LIN {X 0,Y 395.166,Z 181.617,A -85,B 0,C 180,E1 13885.717,E2 13885.717} C_VEL
LIN {X 0,Y 390.867,Z 176.537,A -85,B 0,C 180,E1 13884.321,E2 13884.321} C_VEL
LIN {X 0,Y 388.966,Z 174.114,A -85,B 0,C 180,E1 13883.48,E2 13883.48} C_VEL
LIN {X 0,Y 387.756,Z 171.488,A -85,B 0,C 180,E1 13882.594,E2 13882.594} C_VEL
LIN {X 0,Y 385.429,Z 168.178,A -85,B 0,C 180,E1 13881.136,E2 13881.136} C_VEL
LIN {X 0,Y 384.536,Z 166.163,A -85,B 0,C 180,E1 13880.391,E2 13880.391} C_VEL
LIN {X 0,Y 381.955,Z 162.76,A -85,B 0,C 180,E1 13878.624,E2 13878.624} C_VEL
LIN {X 0,Y 381.043,Z 160.578,A -85,B 0,C 180,E1 13877.721,E2 13877.721} C_VEL
LIN {X 0,Y 378.363,Z 157.325,A -85,B 0,C 180,E1 13875.637,E2 13875.637} C_VEL
LIN {X 0,Y 377.709,Z 155.286,A -85,B 0,C 180,E1 13874.565,E2 13874.565} C_VEL
LIN {X 0,Y 377.671,Z 154.998,A -85,B 0,C 180,E1 13871.762,E2 13871.762} C_VEL
LIN {X 0,Y 377.67,Z 154.99,A -85,B 0,C 180,E1 13867.759,E2 13867.759} C_VEL
LIN {X 0,Y 377.664,Z 154.988,A -85,B 0,C 180,E1 13863.795,E2 13863.795} C_VEL
LIN {X 0,Y 377.658,Z 154.987,A -85,B 0,C 180,E1 13859.848,E2 13859.848} C_VEL
LIN {X 0,Y 377.652,Z 154.988,A -85,B 0,C 180,E1 13855.901,E2 13855.901} C_VEL
LIN {X 0,Y 377.647,Z 154.992,A -85,B 0,C 180,E1 13851.933,E2 13851.933} C_VEL
LIN {X 0,Y 377.647,Z 154.999,A -85,B 0,C 180,E1 13847.927,E2 13847.927} C_VEL
LIN {X 0,Y 377.644,Z 155.008,A -85,B 0,C 180,E1 13843.958,E2 13843.958} C_VEL
LIN {X 0,Y 377.723,Z 155.416,A -85,B 0,C 180,E1 13842.855,E2 13842.855} C_VEL
LIN {X 0,Y 379.411,Z 159.029,A -85,B 0,C 180,E1 13840.927,E2 13840.927} C_VEL
LIN {X 0,Y 381.432,Z 161.353,A -85,B 0,C 180,E1 13839.435,E2 13839.435} C_VEL
LIN {X 0,Y 383.122,Z 164.838,A -85,B 0,C 180,E1 13837.926,E2 13837.926} C_VEL
LIN {X 0,Y 384.74,Z 166.714,A -85,B 0,C 180,E1 13836.895,E2 13836.895} C_VEL
LIN {X 0,Y 386.737,Z 170.482,A -85,B 0,C 180,E1 13835.402,E2 13835.402} C_VEL
LIN {X 0,Y 387.954,Z 172.11,A -85,B 0,C 180,E1 13834.67,E2 13834.67} C_VEL
LIN {X 0,Y 390.476,Z 176.478,A -85,B 0,C 180,E1 13833.049,E2 13833.049} C_VEL
LIN {X 0,Y 394.111,Z 183.067,A -85,B 0,C 180,E1 13830.849,E2 13830.849} C_VEL
LIN {X 0,Y 396.955,Z 188.298,A -85,B 0,C 180,E1 13829.248,E2 13829.248} C_VEL
LIN {X 0,Y 401.414,Z 196.48,A -85,B 0,C 180,E1 13826.941,E2 13826.941} C_VEL
LIN {X 0,Y 408.691,Z 206.89,A -85,B 0,C 180,E1 13824.863,E2 13824.863} C_VEL
LIN {X 0,Y 417.567,Z 219.734,A -85,B 0,C 180,E1 13822.627,E2 13822.627} C_VEL
LIN {X 0,Y 427.427,Z 235.069,A -85,B 0,C 180,E1 13820.355,E2 13820.355} C_VEL
LIN {X 0,Y 431.676,Z 242.453,A -85,B 0,C 180,E1 13819.423,E2 13819.423} C_VEL
LIN {X 0,Y 432.974,Z 254.438,A -85,B 0,C 180,E1 13818.9,E2 13818.9} C_VEL
LIN {X 0,Y 424.415,Z 482.924,A -85,B 0,C 180,E1 13814.793,E2 13814.793} C_VEL
LIN {X 0,Y 422.877,Z 518.615,A -85,B 0,C 180,E1 13814.119,E2 13814.119} C_VEL
LIN {X 0,Y 420.953,Z 540.04,A -85,B 0,C 180,E1 13813.517,E2 13813.517} C_VEL
LIN {X 0,Y 418.413,Z 561.095,A -85,B 0,C 180,E1 13812.691,E2 13812.691} C_VEL
LIN {X 0,Y 415.519,Z 580.617,A -85,B 0,C 180,E1 13811.707,E2 13811.707} C_VEL
LIN {X 0,Y 412.005,Z 600.005,A -85,B 0,C 180,E1 13810.478,E2 13810.478} C_VEL
LIN {X 0,Y 408.151,Z 618.986,A -85,B 0,C 180,E1 13809.018,E2 13809.018} C_VEL
LIN {X 0,Y 404.015,Z 637.17,A -85,B 0,C 180,E1 13807.323,E2 13807.323} C_VEL
LIN {X 0,Y 399.701,Z 654.729,A -85,B 0,C 180,E1 13805.363,E2 13805.363} C_VEL
LIN {X 0,Y 395.442,Z 671.248,A -85,B 0,C 180,E1 13803.183,E2 13803.183} C_VEL
LIN {X 0,Y 392.212,Z 683.238,A -85,B 0,C 180,E1 13801.325,E2 13801.325} C_VEL
LIN {X 0,Y 389.972,Z 688.467,A -85,B 0,C 180,E1 13800.537,E2 13800.537} C_VEL
LIN {X 0,Y 381.254,Z 701.209,A -85,B 0,C 180,E1 13798.63,E2 13798.63} C_VEL
LIN {X 0,Y 379.092,Z 705.741,A -85,B 0,C 180,E1 13797.739,E2 13797.739} C_VEL
LIN {X 0,Y 375.806,Z 717.722,A -85,B 0,C 180,E1 13794.857,E2 13794.857} C_VEL
LIN {X 0,Y 373.033,Z 728.698,A -85,B 0,C 180,E1 13791.708,E2 13791.708} C_VEL
LIN {X 0,Y 370.991,Z 737.873,A -85,B 0,C 180,E1 13788.543,E2 13788.543} C_VEL
LIN {X 0,Y 369.523,Z 745.565,A -85,B 0,C 180,E1 13785.216,E2 13785.216} C_VEL
LIN {X 0,Y 368.595,Z 751.959,A -85,B 0,C 180,E1 13781.69,E2 13781.69} C_VEL
LIN {X 0,Y 368.168,Z 756.552,A -85,B 0,C 180,E1 13778.275,E2 13778.275} C_VEL
LIN {X 0,Y 367.989,Z 759.37,A -85,B 0,C 180,E1 13774.988,E2 13774.988} C_VEL
LIN {X 0,Y 367.942,Z 760.876,A -85,B 0,C 180,E1 13771.557,E2 13771.557} C_VEL
LIN {X 0,Y 367.948,Z 760.909,A -85,B 0,C 180,E1 13768.599,E2 13768.599} C_VEL
LIN {X 0,Y 367.986,Z 759.541,A -85,B 0,C 180,E1 13765.168,E2 13765.168} C_VEL
LIN {X 0,Y 368.12,Z 756.942,A -85,B 0,C 180,E1 13762.038,E2 13762.038} C_VEL
LIN {X 0,Y 368.533,Z 752.507,A -85,B 0,C 180,E1 13758.577,E2 13758.577} C_VEL
LIN {X 0,Y 369.344,Z 746.768,A -85,B 0,C 180,E1 13755.258,E2 13755.258} C_VEL
LIN {X 0,Y 370.692,Z 739.255,A -85,B 0,C 180,E1 13751.93,E2 13751.93} C_VEL
LIN {X 0,Y 372.772,Z 729.787,A -85,B 0,C 180,E1 13748.55,E2 13748.55} C_VEL
LIN {X 0,Y 375.424,Z 719.28,A -85,B 0,C 180,E1 13745.452,E2 13745.452} C_VEL
LIN {X 0,Y 378.7,Z 707.114,A -85,B 0,C 180,E1 13742.482,E2 13742.482} C_VEL
LIN {X 0,Y 382.493,Z 693.534,A -85,B 0,C 180,E1 13739.702,E2 13739.702} C_VEL
LIN {X 0,Y 386.623,Z 679.075,A -85,B 0,C 180,E1 13737.193,E2 13737.193} C_VEL
LIN {X 0,Y 390.999,Z 663.173,A -85,B 0,C 180,E1 13734.876,E2 13734.876} C_VEL
LIN {X 0,Y 395.564,Z 645.973,A -85,B 0,C 180,E1 13732.771,E2 13732.771} C_VEL
LIN {X 0,Y 399.96,Z 628.38,A -85,B 0,C 180,E1 13730.953,E2 13730.953} C_VEL
LIN {X 0,Y 404.219,Z 609.241,A -85,B 0,C 180,E1 13729.325,E2 13729.325} C_VEL
LIN {X 0,Y 408.257,Z 588.889,A -85,B 0,C 180,E1 13727.909,E2 13727.909} C_VEL
LIN {X 0,Y 411.78,Z 568.3,A -85,B 0,C 180,E1 13726.756,E2 13726.756} C_VEL
LIN {X 0,Y 414.498,Z 548.215,A -85,B 0,C 180,E1 13725.889,E2 13725.889} C_VEL
LIN {X 0,Y 416.821,Z 526.068,A -85,B 0,C 180,E1 13725.177,E2 13725.177} C_VEL
LIN {X 0,Y 418.288,Z 503.726,A -85,B 0,C 180,E1 13724.681,E2 13724.681} C_VEL
LIN {X 0,Y 426.979,Z 279.836,A -85,B 0,C 180,E1 13720.629,E2 13720.629} C_VEL
LIN {X 0,Y 427.951,Z 254.162,A -85,B 0,C 180,E1 13720.132,E2 13720.132} C_VEL
LIN {X 0,Y 426.916,Z 246.348,A -85,B 0,C 180,E1 13719.746,E2 13719.746} C_VEL
LIN {X 0,Y 417.063,Z 230.424,A -85,B 0,C 180,E1 13717.469,E2 13717.469} C_VEL
LIN {X 0,Y 407.725,Z 216.316,A -85,B 0,C 180,E1 13715.104,E2 13715.104} C_VEL
LIN {X 0,Y 397.968,Z 202.523,A -85,B 0,C 180,E1 13712.354,E2 13712.354} C_VEL
LIN {X 0,Y 392.606,Z 195.303,A -85,B 0,C 180,E1 13710.62,E2 13710.62} C_VEL
LIN {X 0,Y 390.03,Z 190.525,A -85,B 0,C 180,E1 13709.149,E2 13709.149} C_VEL
LIN {X 0,Y 387.794,Z 186.527,A -85,B 0,C 180,E1 13707.819,E2 13707.819} C_VEL
LIN {X 0,Y 385.711,Z 182.654,A -85,B 0,C 180,E1 13706.479,E2 13706.479} C_VEL
LIN {X 0,Y 382.811,Z 177.599,A -85,B 0,C 180,E1 13704.538,E2 13704.538} C_VEL
LIN {X 0,Y 380.501,Z 173.731,A -85,B 0,C 180,E1 13702.887,E2 13702.887} C_VEL
LIN {X 0,Y 379.69,Z 172.421,A -85,B 0,C 180,E1 13702.285,E2 13702.285} C_VEL
LIN {X 0,Y 377.515,Z 169.146,A -85,B 0,C 180,E1 13700.625,E2 13700.625} C_VEL
LIN {X 0,Y 376.786,Z 167.346,A -85,B 0,C 180,E1 13699.857,E2 13699.857} C_VEL
LIN {X 0,Y 373.937,Z 163.505,A -85,B 0,C 180,E1 13697.426,E2 13697.426} C_VEL
LIN {X 0,Y 373.044,Z 161.554,A -85,B 0,C 180,E1 13696.346,E2 13696.346} C_VEL
LIN {X 0,Y 370.204,Z 157.928,A -85,B 0,C 180,E1 13693.272,E2 13693.272} C_VEL
LIN {X 0,Y 369.725,Z 156.173,A -85,B 0,C 180,E1 13691.861,E2 13691.861} C_VEL
LIN {X 0,Y 369.703,Z 155.98,A -85,B 0,C 180,E1 13687.928,E2 13687.928} C_VEL
LIN {X 0,Y 369.705,Z 155.977,A -85,B 0,C 180,E1 13683.877,E2 13683.877} C_VEL
LIN {X 0,Y 369.708,Z 155.977,A -85,B 0,C 180,E1 13679.845,E2 13679.845} C_VEL
LIN {X 0,Y 369.712,Z 155.982,A -85,B 0,C 180,E1 13675.657,E2 13675.657} C_VEL
LIN {X 0,Y 369.717,Z 155.989,A -85,B 0,C 180,E1 13671.603,E2 13671.603} C_VEL
LIN {X 0,Y 369.788,Z 156.38,A -85,B 0,C 180,E1 13670.192,E2 13670.192} C_VEL
LIN {X 0,Y 371.857,Z 160.462,A -85,B 0,C 180,E1 13667.105,E2 13667.105} C_VEL
LIN {X 0,Y 373.69,Z 162.433,A -85,B 0,C 180,E1 13665.433,E2 13665.433} C_VEL
LIN {X 0,Y 375.581,Z 166.123,A -85,B 0,C 180,E1 13663.45,E2 13663.45} C_VEL
LIN {X 0,Y 377.214,Z 167.9,A -85,B 0,C 180,E1 13662.253,E2 13662.253} C_VEL
LIN {X 0,Y 379.311,Z 171.902,A -85,B 0,C 180,E1 13660.442,E2 13660.442} C_VEL
LIN {X 0,Y 380.668,Z 173.567,A -85,B 0,C 180,E1 13659.554,E2 13659.554} C_VEL
LIN {X 0,Y 382.518,Z 176.962,A -85,B 0,C 180,E1 13658.293,E2 13658.293} C_VEL
LIN {X 0,Y 385.014,Z 179.629,A -85,B 0,C 180,E1 13657.357,E2 13657.357} C_VEL
LIN {X 0,Y 390.258,Z 185.827,A -85,B 0,C 180,E1 13655.518,E2 13655.518} C_VEL
LIN {X 0,Y 394.878,Z 191.397,A -85,B 0,C 180,E1 13654.021,E2 13654.021} C_VEL
LIN {X 0,Y 399.491,Z 197.171,A -85,B 0,C 180,E1 13652.62,E2 13652.62} C_VEL
LIN {X 0,Y 406.598,Z 206.189,A -85,B 0,C 180,E1 13650.621,E2 13650.621} C_VEL
LIN {X 0,Y 417.605,Z 221.402,A -85,B 0,C 180,E1 13647.811,E2 13647.811} C_VEL
LIN {X 0,Y 428.267,Z 237.38,A -85,B 0,C 180,E1 13645.355,E2 13645.355} C_VEL
LIN {X 0,Y 431.593,Z 243.039,A -85,B 0,C 180,E1 13644.622,E2 13644.622} C_VEL
LIN {X 0,Y 421.696,Z 453.338,A -85,B 0,C 180,E1 13640.539,E2 13640.539} C_VEL
LIN {X 0,Y 418.781,Z 513.038,A -85,B 0,C 180,E1 13639.345,E2 13639.345} C_VEL
LIN {X 0,Y 416.496,Z 536.285,A -85,B 0,C 180,E1 13638.676,E2 13638.676} C_VEL
LIN {X 0,Y 413.464,Z 560.266,A -85,B 0,C 180,E1 13637.728,E2 13637.728} C_VEL
LIN {X 0,Y 410.168,Z 581.646,A -85,B 0,C 180,E1 13636.637,E2 13636.637} C_VEL
LIN {X 0,Y 406.403,Z 602.444,A -85,B 0,C 180,E1 13635.316,E2 13635.316} C_VEL
LIN {X 0,Y 402.384,Z 622.536,A -85,B 0,C 180,E1 13633.789,E2 13633.789} C_VEL
LIN {X 0,Y 398.064,Z 641.897,A -85,B 0,C 180,E1 13632.019,E2 13632.019} C_VEL
LIN {X 0,Y 393.619,Z 660.879,A -85,B 0,C 180,E1 13629.989,E2 13629.989} C_VEL
LIN {X 0,Y 389.314,Z 678.385,A -85,B 0,C 180,E1 13627.771,E2 13627.771} C_VEL
LIN {X 0,Y 384.71,Z 696.784,A -85,B 0,C 180,E1 13625.047,E2 13625.047} C_VEL
LIN {X 0,Y 380.795,Z 712.759,A -85,B 0,C 180,E1 13622.277,E2 13622.277} C_VEL
LIN {X 0,Y 377.294,Z 727.194,A -85,B 0,C 180,E1 13619.323,E2 13619.323} C_VEL
LIN {X 0,Y 374.329,Z 740.523,A -85,B 0,C 180,E1 13616.149,E2 13616.149} C_VEL
LIN {X 0,Y 372.125,Z 751.393,A -85,B 0,C 180,E1 13613.096,E2 13613.096} C_VEL
LIN {X 0,Y 370.27,Z 762.065,A -85,B 0,C 180,E1 13609.538,E2 13609.538} C_VEL
LIN {X 0,Y 369.201,Z 769.556,A -85,B 0,C 180,E1 13606.52,E2 13606.52} C_VEL
LIN {X 0,Y 368.446,Z 776.529,A -85,B 0,C 180,E1 13603.017,E2 13603.017} C_VEL
LIN {X 0,Y 368.102,Z 781.139,A -85,B 0,C 180,E1 13600.011,E2 13600.011} C_VEL
LIN {X 0,Y 367.961,Z 784.976,A -85,B 0,C 180,E1 13596.553,E2 13596.553} C_VEL
LIN {X 0,Y 367.926,Z 786.994,A -85,B 0,C 180,E1 13593.427,E2 13593.427} C_VEL
LIN {X 0,Y 367.923,Z 787.81,A -85,B 0,C 180,E1 13590.311,E2 13590.311} C_VEL
LIN {X 0,Y 367.929,Z 787.138,A -85,B 0,C 180,E1 13586.884,E2 13586.884} C_VEL
LIN {X 0,Y 367.952,Z 785.218,A -85,B 0,C 180,E1 13583.76,E2 13583.76} C_VEL
LIN {X 0,Y 368.083,Z 781.58,A -85,B 0,C 180,E1 13580.305,E2 13580.305} C_VEL
LIN {X 0,Y 368.403,Z 777.077,A -85,B 0,C 180,E1 13577.301,E2 13577.301} C_VEL
LIN {X 0,Y 369.11,Z 770.303,A -85,B 0,C 180,E1 13573.799,E2 13573.799} C_VEL
LIN {X 0,Y 370.21,Z 762.431,A -85,B 0,C 180,E1 13570.598,E2 13570.598} C_VEL
LIN {X 0,Y 372.028,Z 751.939,A -85,B 0,C 180,E1 13567.065,E2 13567.065} C_VEL
LIN {X 0,Y 374.196,Z 741.127,A -85,B 0,C 180,E1 13564.011,E2 13564.011} C_VEL
LIN {X 0,Y 377.16,Z 727.779,A -85,B 0,C 180,E1 13560.806,E2 13560.806} C_VEL
LIN {X 0,Y 380.715,Z 713.082,A -85,B 0,C 180,E1 13557.784,E2 13557.784} C_VEL
LIN {X 0,Y 384.475,Z 697.69,A -85,B 0,C 180,E1 13555.102,E2 13555.102} C_VEL
LIN {X 0,Y 388.899,Z 680.083,A -85,B 0,C 180,E1 13552.46,E2 13552.46} C_VEL
LIN {X 0,Y 393.143,Z 662.726,A -85,B 0,C 180,E1 13550.237,E2 13550.237} C_VEL
LIN {X 0,Y 397.724,Z 643.281,A -85,B 0,C 180,E1 13548.121,E2 13548.121} C_VEL
LIN {X 0,Y 402.194,Z 623.378,A -85,B 0,C 180,E1 13546.283,E2 13546.283} C_VEL
LIN {X 0,Y 406.231,Z 603.236,A -85,B 0,C 180,E1 13544.743,E2 13544.743} C_VEL
LIN {X 0,Y 410.06,Z 582.206,A -85,B 0,C 180,E1 13543.398,E2 13543.398} C_VEL
LIN {X 0,Y 413.347,Z 560.902,A -85,B 0,C 180,E1 13542.305,E2 13542.305} C_VEL
LIN {X 0,Y 416.458,Z 536.382,A -85,B 0,C 180,E1 13541.331,E2 13541.331} C_VEL
LIN {X 0,Y 418.745,Z 513.127,A -85,B 0,C 180,E1 13540.661,E2 13540.661} C_VEL
LIN {X 0,Y 421.719,Z 452.113,A -85,B 0,C 180,E1 13539.441,E2 13539.441} C_VEL
LIN {X 0,Y 431.558,Z 242.837,A -85,B 0,C 180,E1 13535.378,E2 13535.378} C_VEL
LIN {X 0,Y 423.08,Z 229.475,A -85,B 0,C 180,E1 13533.492,E2 13533.492} C_VEL
LIN {X 0,Y 413.033,Z 214.984,A -85,B 0,C 180,E1 13531.079,E2 13531.079} C_VEL
LIN {X 0,Y 404.563,Z 203.689,A -85,B 0,C 180,E1 13528.852,E2 13528.852} C_VEL
LIN {X 0,Y 397.353,Z 194.401,A -85,B 0,C 180,E1 13526.77,E2 13526.77} C_VEL
LIN {X 0,Y 392.396,Z 188.417,A -85,B 0,C 180,E1 13525.224,E2 13525.224} C_VEL
LIN {X 0,Y 388.174,Z 183.385,A -85,B 0,C 180,E1 13523.813,E2 13523.813} C_VEL
LIN {X 0,Y 383.503,Z 177.934,A -85,B 0,C 180,E1 13522.131,E2 13522.131} C_VEL
LIN {X 0,Y 381.462,Z 175.518,A -85,B 0,C 180,E1 13521.205,E2 13521.205} C_VEL
LIN {X 0,Y 380.181,Z 172.78,A -85,B 0,C 180,E1 13520.152,E2 13520.152} C_VEL
LIN {X 0,Y 377.689,Z 169.301,A -85,B 0,C 180,E1 13518.362,E2 13518.362} C_VEL
LIN {X 0,Y 376.74,Z 167.247,A -85,B 0,C 180,E1 13517.451,E2 13517.451} C_VEL
LIN {X 0,Y 374.184,Z 163.875,A -85,B 0,C 180,E1 13515.339,E2 13515.339} C_VEL
LIN {X 0,Y 373.131,Z 161.609,A -85,B 0,C 180,E1 13514.113,E2 13514.113} C_VEL
LIN {X 0,Y 370.333,Z 158.146,A -85,B 0,C 180,E1 13511.209,E2 13511.209} C_VEL
LIN {X 0,Y 369.759,Z 156.148,A -85,B 0,C 180,E1 13509.651,E2 13509.651} C_VEL
LIN {X 0,Y 369.738,Z 155.984,A -85,B 0,C 180,E1 13505.586,E2 13505.586} C_VEL
LIN {X 0,Y 369.746,Z 155.991,A -85,B 0,C 180,E1 13501.394,E2 13501.394} C_VEL
LIN {X 0,Y 369.74,Z 155.982,A -85,B 0,C 180,E1 13497.365,E2 13497.365} C_VEL
LIN {X 0,Y 369.751,Z 155.974,A -85,B 0,C 180,E1 13493.166,E2 13493.166} C_VEL
LIN {X 0,Y 369.729,Z 155.975,A -85,B 0,C 180,E1 13489.002,E2 13489.002} C_VEL
LIN {X 0,Y 369.796,Z 156.421,A -85,B 0,C 180,E1 13487.508,E2 13487.508} C_VEL
LIN {X 0,Y 371.777,Z 160.439,A -85,B 0,C 180,E1 13484.558,E2 13484.558} C_VEL
LIN {X 0,Y 373.498,Z 162.115,A -85,B 0,C 180,E1 13483.034,E2 13483.034} C_VEL
LIN {X 0,Y 375.351,Z 165.9,A -85,B 0,C 180,E1 13481.018,E2 13481.018} C_VEL
LIN {X 0,Y 377.132,Z 167.939,A -85,B 0,C 180,E1 13479.677,E2 13479.677} C_VEL
LIN {X 0,Y 379.001,Z 171.688,A -85,B 0,C 180,E1 13477.999,E2 13477.999} C_VEL
LIN {X 0,Y 380.362,Z 173.32,A -85,B 0,C 180,E1 13477.104,E2 13477.104} C_VEL
LIN {X 0,Y 382.66,Z 177.433,A -85,B 0,C 180,E1 13475.405,E2 13475.405} C_VEL
LIN {X 0,Y 383.696,Z 179.193,A -85,B 0,C 180,E1 13474.7,E2 13474.7} C_VEL
LIN {X 0,Y 386.674,Z 184.421,A -85,B 0,C 180,E1 13472.762,E2 13472.762} C_VEL
LIN {X 0,Y 389.597,Z 189.698,A -85,B 0,C 180,E1 13470.984,E2 13470.984} C_VEL
LIN {X 0,Y 392.155,Z 194.438,A -85,B 0,C 180,E1 13469.51,E2 13469.51} C_VEL
LIN {X 0,Y 394.527,Z 198.004,A -85,B 0,C 180,E1 13468.571,E2 13468.571} C_VEL
LIN {X 0,Y 404.508,Z 211.689,A -85,B 0,C 180,E1 13465.65,E2 13465.65} C_VEL
LIN {X 0,Y 414.629,Z 226.73,A -85,B 0,C 180,E1 13463.011,E2 13463.011} C_VEL
LIN {X 0,Y 424.96,Z 243.09,A -85,B 0,C 180,E1 13460.582,E2 13460.582} C_VEL
LIN {X 0,Y 427.049,Z 247.02,A -85,B 0,C 180,E1 13460.105,E2 13460.105} C_VEL
LIN {X 0,Y 427.957,Z 256.049,A -85,B 0,C 180,E1 13459.711,E2 13459.711} C_VEL
LIN {X 0,Y 418.94,Z 484.862,A -85,B 0,C 180,E1 13455.564,E2 13455.564} C_VEL
LIN {X 0,Y 417.374,Z 518.914,A -85,B 0,C 180,E1 13454.911,E2 13454.911} C_VEL
LIN {X 0,Y 415.369,Z 540.34,A -85,B 0,C 180,E1 13454.304,E2 13454.304} C_VEL
LIN {X 0,Y 412.717,Z 561.358,A -85,B 0,C 180,E1 13453.472,E2 13453.472} C_VEL
LIN {X 0,Y 409.609,Z 581.469,A -85,B 0,C 180,E1 13452.448,E2 13452.448} C_VEL
LIN {X 0,Y 405.956,Z 600.706,A -85,B 0,C 180,E1 13451.21,E2 13451.21} C_VEL
LIN {X 0,Y 401.753,Z 620.373,A -85,B 0,C 180,E1 13449.668,E2 13449.668} C_VEL
LIN {X 0,Y 397.464,Z 638.443,A -85,B 0,C 180,E1 13447.955,E2 13447.955} C_VEL
LIN {X 0,Y 393.006,Z 655.66,A -85,B 0,C 180,E1 13445.992,E2 13445.992} C_VEL
LIN {X 0,Y 388.529,Z 672.159,A -85,B 0,C 180,E1 13443.769,E2 13443.769} C_VEL
LIN {X 0,Y 384.293,Z 687.21,A -85,B 0,C 180,E1 13441.356,E2 13441.356} C_VEL
LIN {X 0,Y 380.408,Z 700.921,A -85,B 0,C 180,E1 13438.749,E2 13438.749} C_VEL
LIN {X 0,Y 379.092,Z 705.741,A -85,B 0,C 180,E1 13437.739,E2 13437.739} C_VEL
LIN {X 0,Y 376.959,Z 710.119,A -85,B 0,C 180,E1 13436.816,E2 13436.816} C_VEL
LIN {X 0,Y 368.516,Z 720.971,A -85,B 0,C 180,E1 13434.547,E2 13434.547} C_VEL
LIN {X 0,Y 366.59,Z 724.682,A -85,B 0,C 180,E1 13433.538,E2 13433.538} C_VEL
LIN {X 0,Y 364.042,Z 734.721,A -85,B 0,C 180,E1 13430.246,E2 13430.246} C_VEL
LIN {X 0,Y 362.2,Z 743.207,A -85,B 0,C 180,E1 13426.849,E2 13426.849} C_VEL
LIN {X 0,Y 361.017,Z 749.841,A -85,B 0,C 180,E1 13423.452,E2 13423.452} C_VEL
LIN {X 0,Y 360.343,Z 755.12,A -85,B 0,C 180,E1 13419.906,E2 13419.906} C_VEL
LIN {X 0,Y 360.064,Z 758.667,A -85,B 0,C 180,E1 13416.537,E2 13416.537} C_VEL
LIN {X 0,Y 359.964,Z 760.664,A -85,B 0,C 180,E1 13413.185,E2 13413.185} C_VEL
LIN {X 0,Y 359.952,Z 761.37,A -85,B 0,C 180,E1 13409.823,E2 13409.823} C_VEL
LIN {X 0,Y 359.968,Z 760.573,A -85,B 0,C 180,E1 13406.497,E2 13406.497} C_VEL
LIN {X 0,Y 360.081,Z 758.301,A -85,B 0,C 180,E1 13402.982,E2 13402.982} C_VEL
LIN {X 0,Y 360.367,Z 754.841,A -85,B 0,C 180,E1 13399.772,E2 13399.772} C_VEL
LIN {X 0,Y 361.082,Z 749.428,A -85,B 0,C 180,E1 13396.224,E2 13396.224} C_VEL
LIN {X 0,Y 362.308,Z 742.685,A -85,B 0,C 180,E1 13392.826,E2 13392.826} C_VEL
LIN {X 0,Y 364.212,Z 734.045,A -85,B 0,C 180,E1 13389.413,E2 13389.413} C_VEL
LIN {X 0,Y 366.741,Z 724.114,A -85,B 0,C 180,E1 13386.204,E2 13386.204} C_VEL
LIN {X 0,Y 369.976,Z 712.627,A -85,B 0,C 180,E1 13383.104,E2 13383.104} C_VEL
LIN {X 0,Y 373.6,Z 700.227,A -85,B 0,C 180,E1 13380.324,E2 13380.324} C_VEL
LIN {X 0,Y 378.004,Z 685.418,A -85,B 0,C 180,E1 13377.524,E2 13377.524} C_VEL
LIN {X 0,Y 382.562,Z 670.106,A -85,B 0,C 180,E1 13375.085,E2 13375.085} C_VEL
LIN {X 0,Y 387.044,Z 654.195,A -85,B 0,C 180,E1 13372.963,E2 13372.963} C_VEL
LIN {X 0,Y 392.055,Z 635.422,A -85,B 0,C 180,E1 13370.863,E2 13370.863} C_VEL
LIN {X 0,Y 396.646,Z 616.823,A -85,B 0,C 180,E1 13369.134,E2 13369.134} C_VEL
LIN {X 0,Y 400.827,Z 597.451,A -85,B 0,C 180,E1 13367.663,E2 13367.663} C_VEL
LIN {X 0,Y 404.786,Z 576.315,A -85,B 0,C 180,E1 13366.364,E2 13366.364} C_VEL
LIN {X 0,Y 408.071,Z 555.322,A -85,B 0,C 180,E1 13365.347,E2 13365.347} C_VEL
LIN {X 0,Y 410.579,Z 534.464,A -85,B 0,C 180,E1 13364.597,E2 13364.597} C_VEL
LIN {X 0,Y 412.508,Z 511.375,A -85,B 0,C 180,E1 13364.013,E2 13364.013} C_VEL
LIN {X 0,Y 421.76,Z 287.062,A -85,B 0,C 180,E1 13359.904,E2 13359.904} C_VEL
LIN {X 0,Y 423.033,Z 255.87,A -85,B 0,C 180,E1 13359.304,E2 13359.304} C_VEL
LIN {X 0,Y 422.307,Z 250.816,A -85,B 0,C 180,E1 13359.034,E2 13359.034} C_VEL
LIN {X 0,Y 412.164,Z 234.313,A -85,B 0,C 180,E1 13356.596,E2 13356.596} C_VEL
LIN {X 0,Y 403.507,Z 221.329,A -85,B 0,C 180,E1 13354.314,E2 13354.314} C_VEL
LIN {X 0,Y 395.293,Z 209.44,A -85,B 0,C 180,E1 13351.914,E2 13351.914} C_VEL
LIN {X 0,Y 386.834,Z 198.228,A -85,B 0,C 180,E1 13349.158,E2 13349.158} C_VEL
LIN {X 0,Y 383.857,Z 193.883,A -85,B 0,C 180,E1 13347.96,E2 13347.96} C_VEL
LIN {X 0,Y 380.77,Z 188.523,A -85,B 0,C 180,E1 13346.01,E2 13346.01} C_VEL
LIN {X 0,Y 378.416,Z 184.172,A -85,B 0,C 180,E1 13344.343,E2 13344.343} C_VEL
LIN {X 0,Y 376.141,Z 180.315,A -85,B 0,C 180,E1 13342.671,E2 13342.671} C_VEL
LIN {X 0,Y 375.196,Z 178.887,A -85,B 0,C 180,E1 13341.973,E2 13341.973} C_VEL
LIN {X 0,Y 373.095,Z 175.329,A -85,B 0,C 180,E1 13340.225,E2 13340.225} C_VEL
LIN {X 0,Y 372.382,Z 173.915,A -85,B 0,C 180,E1 13339.538,E2 13339.538} C_VEL
LIN {X 0,Y 369.75,Z 170.073,A -85,B 0,C 180,E1 13337.143,E2 13337.143} C_VEL
LIN {X 0,Y 368.992,Z 168.429,A -85,B 0,C 180,E1 13336.207,E2 13336.207} C_VEL
LIN {X 0,Y 366.145,Z 164.537,A -85,B 0,C 180,E1 13332.94,E2 13332.94} C_VEL
LIN {X 0,Y 365.359,Z 162.745,A -85,B 0,C 180,E1 13331.524,E2 13331.524} C_VEL
LIN {X 0,Y 362.162,Z 158.598,A -85,B 0,C 180,E1 13324.275,E2 13324.275} C_VEL
LIN {X 0,Y 362.001,Z 157.968,A -85,B 0,C 180,E1 13320.633,E2 13320.633} C_VEL
LIN {X 0,Y 362.394,Z 159.146,A -85,B 0,C 180,E1 13316.837,E2 13316.837} C_VEL
LIN {X 0,Y 365.714,Z 163.154,A -85,B 0,C 180,E1 13310.4,E2 13310.4} C_VEL
LIN {X 0,Y 368.014,Z 167.484,A -85,B 0,C 180,E1 13307.128,E2 13307.128} C_VEL
LIN {X 0,Y 369.652,Z 169.302,A -85,B 0,C 180,E1 13305.591,E2 13305.591} C_VEL
LIN {X 0,Y 371.525,Z 172.963,A -85,B 0,C 180,E1 13303.586,E2 13303.586} C_VEL
LIN {X 0,Y 373.084,Z 174.856,A -85,B 0,C 180,E1 13302.372,E2 13302.372} C_VEL
LIN {X 0,Y 374.939,Z 178.202,A -85,B 0,C 180,E1 13300.933,E2 13300.933} C_VEL
LIN {X 0,Y 377.718,Z 181.017,A -85,B 0,C 180,E1 13299.751,E2 13299.751} C_VEL
LIN {X 0,Y 382.978,Z 187.146,A -85,B 0,C 180,E1 13297.675,E2 13297.675} C_VEL
LIN {X 0,Y 388.056,Z 193.22,A -85,B 0,C 180,E1 13295.856,E2 13295.856} C_VEL
LIN {X 0,Y 392.51,Z 198.672,A -85,B 0,C 180,E1 13294.38,E2 13294.38} C_VEL
LIN {X 0,Y 397.062,Z 204.459,A -85,B 0,C 180,E1 13292.966,E2 13292.966} C_VEL
LIN {X 0,Y 403.962,Z 213.404,A -85,B 0,C 180,E1 13290.98,E2 13290.98} C_VEL
LIN {X 0,Y 414.23,Z 227.759,A -85,B 0,C 180,E1 13288.292,E2 13288.292} C_VEL
LIN {X 0,Y 424.679,Z 243.653,A -85,B 0,C 180,E1 13285.819,E2 13285.819} C_VEL
LIN {X 0,Y 426.518,Z 246.843,A -85,B 0,C 180,E1 13285.399,E2 13285.399} C_VEL
LIN {X 0,Y 416.251,Z 456.154,A -85,B 0,C 180,E1 13281.306,E2 13281.306} C_VEL
LIN {X 0,Y 413.336,Z 513.226,A -85,B 0,C 180,E1 13280.153,E2 13280.153} C_VEL
LIN {X 0,Y 410.967,Z 536.474,A -85,B 0,C 180,E1 13279.48,E2 13279.48} C_VEL
LIN {X 0,Y 407.761,Z 560.767,A -85,B 0,C 180,E1 13278.511,E2 13278.511} C_VEL
LIN {X 0,Y 404.329,Z 582.137,A -85,B 0,C 180,E1 13277.41,E2 13277.41} C_VEL
LIN {X 0,Y 400.42,Z 602.772,A -85,B 0,C 180,E1 13276.084,E2 13276.084} C_VEL
LIN {X 0,Y 396.103,Z 623.414,A -85,B 0,C 180,E1 13274.493,E2 13274.493} C_VEL
LIN {X 0,Y 391.445,Z 643.275,A -85,B 0,C 180,E1 13272.64,E2 13272.64} C_VEL
LIN {X 0,Y 386.418,Z 663.495,A -85,B 0,C 180,E1 13270.402,E2 13270.402} C_VEL
LIN {X 0,Y 381.908,Z 681.075,A -85,B 0,C 180,E1 13268.105,E2 13268.105} C_VEL
LIN {X 0,Y 377.351,Z 698.199,A -85,B 0,C 180,E1 13265.469,E2 13265.469} C_VEL
LIN {X 0,Y 373.181,Z 714.266,A -85,B 0,C 180,E1 13262.583,E2 13262.583} C_VEL
LIN {X 0,Y 369.659,Z 728.079,A -85,B 0,C 180,E1 13259.668,E2 13259.668} C_VEL
LIN {X 0,Y 366.395,Z 741.904,A -85,B 0,C 180,E1 13256.236,E2 13256.236} C_VEL
LIN {X 0,Y 364.041,Z 753.129,A -85,B 0,C 180,E1 13252.954,E2 13252.954} C_VEL
LIN {X 0,Y 362.251,Z 762.854,A -85,B 0,C 180,E1 13249.51,E2 13249.51} C_VEL
LIN {X 0,Y 361.074,Z 770.939,A -85,B 0,C 180,E1 13246.076,E2 13246.076} C_VEL
LIN {X 0,Y 360.418,Z 776.965,A -85,B 0,C 180,E1 13242.822,E2 13242.822} C_VEL
LIN {X 0,Y 360.068,Z 781.886,A -85,B 0,C 180,E1 13239.429,E2 13239.429} C_VEL
LIN {X 0,Y 359.949,Z 785.151,A -85,B 0,C 180,E1 13236.045,E2 13236.045} C_VEL
LIN {X 0,Y 359.932,Z 786.911,A -85,B 0,C 180,E1 13233.025,E2 13233.025} C_VEL
LIN {X 0,Y 359.926,Z 787.497,A -85,B 0,C 180,E1 13229.523,E2 13229.523} C_VEL
LIN {X 0,Y 359.931,Z 786.701,A -85,B 0,C 180,E1 13226.496,E2 13226.496} C_VEL
LIN {X 0,Y 359.972,Z 784.545,A -85,B 0,C 180,E1 13223.141,E2 13223.141} C_VEL
LIN {X 0,Y 360.121,Z 780.807,A -85,B 0,C 180,E1 13219.765,E2 13219.765} C_VEL
LIN {X 0,Y 360.487,Z 776.163,A -85,B 0,C 180,E1 13216.691,E2 13216.691} C_VEL
LIN {X 0,Y 361.306,Z 769.135,A -85,B 0,C 180,E1 13213.108,E2 13213.108} C_VEL
LIN {X 0,Y 362.539,Z 761.153,A -85,B 0,C 180,E1 13209.835,E2 13209.835} C_VEL
LIN {X 0,Y 364.448,Z 750.979,A -85,B 0,C 180,E1 13206.388,E2 13206.388} C_VEL
LIN {X 0,Y 366.958,Z 739.51,A -85,B 0,C 180,E1 13203.109,E2 13203.109} C_VEL
LIN {X 0,Y 370.01,Z 726.615,A -85,B 0,C 180,E1 13200.007,E2 13200.007} C_VEL
LIN {X 0,Y 373.611,Z 712.63,A -85,B 0,C 180,E1 13197.095,E2 13197.095} C_VEL
LIN {X 0,Y 377.735,Z 696.746,A -85,B 0,C 180,E1 13194.293,E2 13194.293} C_VEL
LIN {X 0,Y 382.554,Z 678.435,A -85,B 0,C 180,E1 13191.536,E2 13191.536} C_VEL
LIN {X 0,Y 387.242,Z 660.33,A -85,B 0,C 180,E1 13189.215,E2 13189.215} C_VEL
LIN {X 0,Y 391.906,Z 641.273,A -85,B 0,C 180,E1 13187.165,E2 13187.165} C_VEL
LIN {X 0,Y 396.609,Z 620.894,A -85,B 0,C 180,E1 13185.304,E2 13185.304} C_VEL
LIN {X 0,Y 400.618,Z 601.661,A -85,B 0,C 180,E1 13183.841,E2 13183.841} C_VEL
LIN {X 0,Y 404.901,Z 578.424,A -85,B 0,C 180,E1 13182.387,E2 13182.387} C_VEL
LIN {X 0,Y 408.452,Z 556.166,A -85,B 0,C 180,E1 13181.28,E2 13181.28} C_VEL
LIN {X 0,Y 411.263,Z 533.672,A -85,B 0,C 180,E1 13180.433,E2 13180.433} C_VEL
LIN {X 0,Y 413.541,Z 509.555,A -85,B 0,C 180,E1 13179.771,E2 13179.771} C_VEL
LIN {X 0,Y 422.734,Z 321.79,A -85,B 0,C 180,E1 13176.065,E2 13176.065} C_VEL
LIN {X 0,Y 426.372,Z 246.372,A -85,B 0,C 180,E1 13174.576,E2 13174.576} C_VEL
LIN {X 0,Y 415.775,Z 230.03,A -85,B 0,C 180,E1 13172.104,E2 13172.104} C_VEL
LIN {X 0,Y 405.964,Z 216.185,A -85,B 0,C 180,E1 13169.591,E2 13169.591} C_VEL
LIN {X 0,Y 398.177,Z 205.904,A -85,B 0,C 180,E1 13167.397,E2 13167.397} C_VEL
LIN {X 0,Y 393.882,Z 200.43,A -85,B 0,C 180,E1 13166.09,E2 13166.09} C_VEL
LIN {X 0,Y 389.862,Z 195.426,A -85,B 0,C 180,E1 13164.791,E2 13164.791} C_VEL
LIN {X 0,Y 385.71,Z 190.418,A -85,B 0,C 180,E1 13163.366,E2 13163.366} C_VEL
LIN {X 0,Y 381.403,Z 185.289,A -85,B 0,C 180,E1 13161.774,E2 13161.774} C_VEL
LIN {X 0,Y 376.491,Z 179.652,A -85,B 0,C 180,E1 13159.792,E2 13159.792} C_VEL
LIN {X 0,Y 373.937,Z 176.877,A -85,B 0,C 180,E1 13158.553,E2 13158.553} C_VEL
LIN {X 0,Y 372.668,Z 174.094,A -85,B 0,C 180,E1 13157.326,E2 13157.326} C_VEL
LIN {X 0,Y 370.14,Z 170.733,A -85,B 0,C 180,E1 13155.19,E2 13155.19} C_VEL
LIN {X 0,Y 369.101,Z 168.475,A -85,B 0,C 180,E1 13153.951,E2 13153.951} C_VEL
LIN {X 0,Y 366.373,Z 164.982,A -85,B 0,C 180,E1 13151.013,E2 13151.013} C_VEL
LIN {X 0,Y 365.375,Z 162.708,A -85,B 0,C 180,E1 13149.291,E2 13149.291} C_VEL
LIN {X 0,Y 362.042,Z 158.18,A -85,B 0,C 180,E1 13141.582,E2 13141.582} C_VEL
LIN {X 0,Y 361.897,Z 157.705,A -85,B 0,C 180,E1 13138.258,E2 13138.258} C_VEL
LIN {X 0,Y 362.224,Z 158.799,A -85,B 0,C 180,E1 13134.615,E2 13134.615} C_VEL
LIN {X 0,Y 365.732,Z 163.223,A -85,B 0,C 180,E1 13127.687,E2 13127.687} C_VEL
LIN {X 0,Y 367.907,Z 167.468,A -85,B 0,C 180,E1 13124.554,E2 13124.554} C_VEL
LIN {X 0,Y 369.43,Z 169.005,A -85,B 0,C 180,E1 13123.166,E2 13123.166} C_VEL
LIN {X 0,Y 371.437,Z 172.951,A -85,B 0,C 180,E1 13120.991,E2 13120.991} C_VEL
LIN {X 0,Y 372.841,Z 174.521,A -85,B 0,C 180,E1 13119.924,E2 13119.924} C_VEL
LIN {X 0,Y 374.666,Z 178.273,A -85,B 0,C 180,E1 13118.226,E2 13118.226} C_VEL
LIN {X 0,Y 375.997,Z 179.916,A -85,B 0,C 180,E1 13117.32,E2 13117.32} C_VEL
LIN {X 0,Y 378.445,Z 184.212,A -85,B 0,C 180,E1 13115.493,E2 13115.493} C_VEL
LIN {X 0,Y 382.208,Z 191.032,A -85,B 0,C 180,E1 13112.923,E2 13112.923} C_VEL
LIN {X 0,Y 384.979,Z 195.728,A -85,B 0,C 180,E1 13111.368,E2 13111.368} C_VEL
LIN {X 0,Y 392.622,Z 206.028,A -85,B 0,C 180,E1 13108.786,E2 13108.786} C_VEL
LIN {X 0,Y 399.669,Z 215.74,A -85,B 0,C 180,E1 13106.654,E2 13106.654} C_VEL
LIN {X 0,Y 408.937,Z 229.457,A -85,B 0,C 180,E1 13104.112,E2 13104.112} C_VEL
LIN {X 0,Y 418.727,Z 244.89,A -85,B 0,C 180,E1 13101.688,E2 13101.688} C_VEL
LIN {X 0,Y 422.492,Z 251.627,A -85,B 0,C 180,E1 13100.8,E2 13100.8} C_VEL
LIN {X 0,Y 423.016,Z 257.885,A -85,B 0,C 180,E1 13100.538,E2 13100.538} C_VEL
LIN {X 0,Y 413.54,Z 486.808,A -85,B 0,C 180,E1 13096.354,E2 13096.354} C_VEL
LIN {X 0,Y 411.937,Z 519.356,A -85,B 0,C 180,E1 13095.72,E2 13095.72} C_VEL
LIN {X 0,Y 409.851,Z 540.752,A -85,B 0,C 180,E1 13095.109,E2 13095.109} C_VEL
LIN {X 0,Y 407.099,Z 561.605,A -85,B 0,C 180,E1 13094.276,E2 13094.276} C_VEL
LIN {X 0,Y 403.762,Z 582.241,A -85,B 0,C 180,E1 13093.211,E2 13093.211} C_VEL
LIN {X 0,Y 399.975,Z 601.395,A -85,B 0,C 180,E1 13091.965,E2 13091.965} C_VEL
LIN {X 0,Y 395.407,Z 621.748,A -85,B 0,C 180,E1 13090.34,E2 13090.34} C_VEL
LIN {X 0,Y 390.833,Z 640.188,A -85,B 0,C 180,E1 13088.556,E2 13088.556} C_VEL
LIN {X 0,Y 386.156,Z 657.328,A -85,B 0,C 180,E1 13086.549,E2 13086.549} C_VEL
LIN {X 0,Y 381.2,Z 674.566,A -85,B 0,C 180,E1 13084.145,E2 13084.145} C_VEL
LIN {X 0,Y 376.846,Z 689.402,A -85,B 0,C 180,E1 13081.69,E2 13081.69} C_VEL
LIN {X 0,Y 372.821,Z 702.805,A -85,B 0,C 180,E1 13079.038,E2 13079.038} C_VEL
LIN {X 0,Y 369.085,Z 715.651,A -85,B 0,C 180,E1 13076.03,E2 13076.03} C_VEL
LIN {X 0,Y 366.59,Z 724.682,A -85,B 0,C 180,E1 13073.538,E2 13073.538} C_VEL
LIN {X 0,Y 364.725,Z 728.34,A -85,B 0,C 180,E1 13072.504,E2 13072.504} C_VEL
LIN {X 0,Y 356.513,Z 737.486,A -85,B 0,C 180,E1 13069.746,E2 13069.746} C_VEL
LIN {X 0,Y 355.181,Z 739.967,A -85,B 0,C 180,E1 13068.774,E2 13068.774} C_VEL
LIN {X 0,Y 353.6,Z 747.562,A -85,B 0,C 180,E1 13065.246,E2 13065.246} C_VEL
LIN {X 0,Y 352.655,Z 753.239,A -85,B 0,C 180,E1 13061.779,E2 13061.779} C_VEL
LIN {X 0,Y 352.174,Z 757.61,A -85,B 0,C 180,E1 13058.161,E2 13058.161} C_VEL
LIN {X 0,Y 352.003,Z 760.178,A -85,B 0,C 180,E1 13054.888,E2 13054.888} C_VEL
LIN {X 0,Y 351.954,Z 761.5,A -85,B 0,C 180,E1 13051.302,E2 13051.302} C_VEL
LIN {X 0,Y 351.958,Z 761.428,A -85,B 0,C 180,E1 13048.046,E2 13048.046} C_VEL
LIN {X 0,Y 352.013,Z 759.918,A -85,B 0,C 180,E1 13044.622,E2 13044.622} C_VEL
LIN {X 0,Y 352.226,Z 757.091,A -85,B 0,C 180,E1 13041.183,E2 13041.183} C_VEL
LIN {X 0,Y 352.743,Z 752.65,A -85,B 0,C 180,E1 13037.726,E2 13037.726} C_VEL
LIN {X 0,Y 353.807,Z 746.411,A -85,B 0,C 180,E1 13034.091,E2 13034.091} C_VEL
LIN {X 0,Y 355.49,Z 738.761,A -85,B 0,C 180,E1 13030.617,E2 13030.617} C_VEL
LIN {X 0,Y 357.904,Z 729.329,A -85,B 0,C 180,E1 13027.207,E2 13027.207} C_VEL
LIN {X 0,Y 361.284,Z 717.565,A -85,B 0,C 180,E1 13023.718,E2 13023.718} C_VEL
LIN {X 0,Y 364.919,Z 705.817,A -85,B 0,C 180,E1 13020.811,E2 13020.811} C_VEL
LIN {X 0,Y 369.276,Z 691.827,A -85,B 0,C 180,E1 13017.939,E2 13017.939} C_VEL
LIN {X 0,Y 374.051,Z 676.495,A -85,B 0,C 180,E1 13015.295,E2 13015.295} C_VEL
LIN {X 0,Y 378.864,Z 660.789,A -85,B 0,C 180,E1 13013.008,E2 13013.008} C_VEL
LIN {X 0,Y 383.774,Z 643.507,A -85,B 0,C 180,E1 13010.915,E2 13010.915} C_VEL
LIN {X 0,Y 388.742,Z 624.729,A -85,B 0,C 180,E1 13009.016,E2 13009.016} C_VEL
LIN {X 0,Y 393.269,Z 606.017,A -85,B 0,C 180,E1 13007.447,E2 13007.447} C_VEL
LIN {X 0,Y 397.349,Z 586.356,A -85,B 0,C 180,E1 13006.114,E2 13006.114} C_VEL
LIN {X 0,Y 401.16,Z 564.789,A -85,B 0,C 180,E1 13004.942,E2 13004.942} C_VEL
LIN {X 0,Y 404.113,Z 544.159,A -85,B 0,C 180,E1 13004.075,E2 13004.075} C_VEL
LIN {X 0,Y 406.388,Z 522.408,A -85,B 0,C 180,E1 13003.421,E2 13003.421} C_VEL
LIN {X 0,Y 408.031,Z 494.489,A -85,B 0,C 180,E1 13002.845,E2 13002.845} C_VEL
LIN {X 0,Y 417.838,Z 267.785,A -85,B 0,C 180,E1 12998.669,E2 12998.669} C_VEL
LIN {X 0,Y 418.189,Z 257.38,A -85,B 0,C 180,E1 12998.447,E2 12998.447} C_VEL
LIN {X 0,Y 417.766,Z 255.249,A -85,B 0,C 180,E1 12998.307,E2 12998.307} C_VEL
LIN {X 0,Y 407.47,Z 238.461,A -85,B 0,C 180,E1 12995.733,E2 12995.733} C_VEL
LIN {X 0,Y 397.606,Z 223.529,A -85,B 0,C 180,E1 12992.986,E2 12992.986} C_VEL
LIN {X 0,Y 391.153,Z 214.511,A -85,B 0,C 180,E1 12991.002,E2 12991.002} C_VEL
LIN {X 0,Y 385.047,Z 206.014,A -85,B 0,C 180,E1 12988.937,E2 12988.937} C_VEL
LIN {X 0,Y 380.66,Z 200.288,A -85,B 0,C 180,E1 12987.323,E2 12987.323} C_VEL
LIN {X 0,Y 375.369,Z 193.388,A -85,B 0,C 180,E1 12985.142,E2 12985.142} C_VEL
LIN {X 0,Y 373.788,Z 190.449,A -85,B 0,C 180,E1 12983.991,E2 12983.991} C_VEL
LIN {X 0,Y 371.223,Z 185.877,A -85,B 0,C 180,E1 12981.987,E2 12981.987} C_VEL
LIN {X 0,Y 368.95,Z 182.276,A -85,B 0,C 180,E1 12980.131,E2 12980.131} C_VEL
LIN {X 0,Y 368.181,Z 180.651,A -85,B 0,C 180,E1 12979.349,E2 12979.349} C_VEL
LIN {X 0,Y 365.575,Z 176.641,A -85,B 0,C 180,E1 12976.853,E2 12976.853} C_VEL
LIN {X 0,Y 364.946,Z 175.303,A -85,B 0,C 180,E1 12976.064,E2 12976.064} C_VEL
LIN {X 0,Y 362.175,Z 171.39,A -85,B 0,C 180,E1 12972.76,E2 12972.76} C_VEL
LIN {X 0,Y 361.386,Z 169.657,A -85,B 0,C 180,E1 12971.329,E2 12971.329} C_VEL
LIN {X 0,Y 358.408,Z 165.68,A -85,B 0,C 180,E1 12964.32,E2 12964.32} C_VEL
LIN {X 0,Y 358.241,Z 165.031,A -85,B 0,C 180,E1 12960.64,E2 12960.64} C_VEL
LIN {X 0,Y 358.646,Z 166.24,A -85,B 0,C 180,E1 12956.804,E2 12956.804} C_VEL
LIN {X 0,Y 361.871,Z 170.191,A -85,B 0,C 180,E1 12950.458,E2 12950.458} C_VEL
LIN {X 0,Y 364.004,Z 174.344,A -85,B 0,C 180,E1 12947.306,E2 12947.306} C_VEL
LIN {X 0,Y 365.611,Z 176.173,A -85,B 0,C 180,E1 12945.752,E2 12945.752} C_VEL
LIN {X 0,Y 367.254,Z 179.348,A -85,B 0,C 180,E1 12944.121,E2 12944.121} C_VEL
LIN {X 0,Y 370.188,Z 182.153,A -85,B 0,C 180,E1 12942.635,E2 12942.635} C_VEL
LIN {X 0,Y 375.127,Z 187.567,A -85,B 0,C 180,E1 12940.377,E2 12940.377} C_VEL
LIN {X 0,Y 379.985,Z 193.252,A -85,B 0,C 180,E1 12938.384,E2 12938.384} C_VEL
LIN {X 0,Y 386.55,Z 201.475,A -85,B 0,C 180,E1 12935.959,E2 12935.959} C_VEL
LIN {X 0,Y 390.362,Z 206.214,A -85,B 0,C 180,E1 12934.676,E2 12934.676} C_VEL
LIN {X 0,Y 394.968,Z 212.159,A -85,B 0,C 180,E1 12933.218,E2 12933.218} C_VEL
LIN {X 0,Y 401.906,Z 221.409,A -85,B 0,C 180,E1 12931.183,E2 12931.183} C_VEL
LIN {X 0,Y 411.248,Z 234.662,A -85,B 0,C 180,E1 12928.689,E2 12928.689} C_VEL
LIN {X 0,Y 421.374,Z 250.333,A -85,B 0,C 180,E1 12926.232,E2 12926.232} C_VEL
LIN {X 0,Y 421.368,Z 253.664,A -85,B 0,C 180,E1 12926.136,E2 12926.136} C_VEL
LIN {X 0,Y 410.748,Z 461.783,A -85,B 0,C 180,E1 12922.038,E2 12922.038} C_VEL
LIN {X 0,Y 407.959,Z 513.614,A -85,B 0,C 180,E1 12920.978,E2 12920.978} C_VEL
LIN {X 0,Y 405.509,Z 536.795,A -85,B 0,C 180,E1 12920.302,E2 12920.302} C_VEL
LIN {X 0,Y 402.338,Z 560.02,A -85,B 0,C 180,E1 12919.376,E2 12919.376} C_VEL
LIN {X 0,Y 398.914,Z 580.564,A -85,B 0,C 180,E1 12918.323,E2 12918.323} C_VEL
LIN {X 0,Y 394.729,Z 602.061,A -85,B 0,C 180,E1 12916.95,E2 12916.95} C_VEL
LIN {X 0,Y 390.364,Z 622.155,A -85,B 0,C 180,E1 12915.401,E2 12915.401} C_VEL
LIN {X 0,Y 385.66,Z 641.525,A -85,B 0,C 180,E1 12913.599,E2 12913.599} C_VEL
LIN {X 0,Y 380.882,Z 660.164,A -85,B 0,C 180,E1 12911.569,E2 12911.569} C_VEL
LIN {X 0,Y 376.017,Z 677.983,A -85,B 0,C 180,E1 12909.26,E2 12909.26} C_VEL
LIN {X 0,Y 370.945,Z 696.32,A -85,B 0,C 180,E1 12906.465,E2 12906.465} C_VEL
LIN {X 0,Y 366.565,Z 712.207,A -85,B 0,C 180,E1 12903.621,E2 12903.621} C_VEL
LIN {X 0,Y 362.752,Z 726.212,A -85,B 0,C 180,E1 12900.657,E2 12900.657} C_VEL
LIN {X 0,Y 359.46,Z 739.238,A -85,B 0,C 180,E1 12897.463,E2 12897.463} C_VEL
LIN {X 0,Y 356.799,Z 750.587,A -85,B 0,C 180,E1 12894.15,E2 12894.15} C_VEL
LIN {X 0,Y 354.668,Z 761.204,A -85,B 0,C 180,E1 12890.461,E2 12890.461} C_VEL
LIN {X 0,Y 353.42,Z 768.764,A -85,B 0,C 180,E1 12887.28,E2 12887.28} C_VEL
LIN {X 0,Y 352.536,Z 775.803,A -85,B 0,C 180,E1 12883.615,E2 12883.615} C_VEL
LIN {X 0,Y 352.144,Z 780.46,A -85,B 0,C 180,E1 12880.47,E2 12880.47} C_VEL
LIN {X 0,Y 351.974,Z 784.354,A -85,B 0,C 180,E1 12876.852,E2 12876.852} C_VEL
LIN {X 0,Y 351.936,Z 786.401,A -85,B 0,C 180,E1 12873.583,E2 12873.583} C_VEL
LIN {X 0,Y 351.933,Z 787.229,A -85,B 0,C 180,E1 12870.326,E2 12870.326} C_VEL
LIN {X 0,Y 351.937,Z 786.617,A -85,B 0,C 180,E1 12866.906,E2 12866.906} C_VEL
LIN {X 0,Y 351.956,Z 784.835,A -85,B 0,C 180,E1 12863.803,E2 12863.803} C_VEL
LIN {X 0,Y 352.081,Z 781.548,A -85,B 0,C 180,E1 12860.355,E2 12860.355} C_VEL
LIN {X 0,Y 352.457,Z 776.608,A -85,B 0,C 180,E1 12856.883,E2 12856.883} C_VEL
LIN {X 0,Y 353.221,Z 770.243,A -85,B 0,C 180,E1 12853.388,E2 12853.388} C_VEL
LIN {X 0,Y 354.521,Z 762.054,A -85,B 0,C 180,E1 12849.875,E2 12849.875} C_VEL
LIN {X 0,Y 356.472,Z 752.203,A -85,B 0,C 180,E1 12846.354,E2 12846.354} C_VEL
LIN {X 0,Y 358.89,Z 741.51,A -85,B 0,C 180,E1 12843.172,E2 12843.172} C_VEL
LIN {X 0,Y 362.369,Z 727.659,A -85,B 0,C 180,E1 12839.674,E2 12839.674} C_VEL
LIN {X 0,Y 366.148,Z 713.696,A -85,B 0,C 180,E1 12836.679,E2 12836.679} C_VEL
LIN {X 0,Y 370.534,Z 697.733,A -85,B 0,C 180,E1 12833.776,E2 12833.776} C_VEL
LIN {X 0,Y 375.262,Z 680.81,A -85,B 0,C 180,E1 12831.137,E2 12831.137} C_VEL
LIN {X 0,Y 380.015,Z 663.176,A -85,B 0,C 180,E1 12828.807,E2 12828.807} C_VEL
LIN {X 0,Y 385.274,Z 642.966,A -85,B 0,C 180,E1 12826.551,E2 12826.551} C_VEL
LIN {X 0,Y 389.955,Z 623.829,A -85,B 0,C 180,E1 12824.747,E2 12824.747} C_VEL
LIN {X 0,Y 394.372,Z 603.659,A -85,B 0,C 180,E1 12823.17,E2 12823.17} C_VEL
LIN {X 0,Y 398.578,Z 582.395,A -85,B 0,C 180,E1 12821.785,E2 12821.785} C_VEL
LIN {X 0,Y 402.127,Z 561.143,A -85,B 0,C 180,E1 12820.682,E2 12820.682} C_VEL
LIN {X 0,Y 405.485,Z 536.701,A -85,B 0,C 180,E1 12819.7,E2 12819.7} C_VEL
LIN {X 0,Y 407.937,Z 513.435,A -85,B 0,C 180,E1 12819.022,E2 12819.022} C_VEL
LIN {X 0,Y 410.916,Z 457.548,A -85,B 0,C 180,E1 12817.884,E2 12817.884} C_VEL
LIN {X 0,Y 421.469,Z 250.554,A -85,B 0,C 180,E1 12813.809,E2 12813.809} C_VEL
LIN {X 0,Y 411.432,Z 234.977,A -85,B 0,C 180,E1 12811.377,E2 12811.377} C_VEL
LIN {X 0,Y 402.178,Z 221.814,A -85,B 0,C 180,E1 12808.917,E2 12808.917} C_VEL
LIN {X 0,Y 395.099,Z 212.351,A -85,B 0,C 180,E1 12806.854,E2 12806.854} C_VEL
LIN {X 0,Y 388.365,Z 203.537,A -85,B 0,C 180,E1 12804.69,E2 12804.69} C_VEL
LIN {X 0,Y 382.983,Z 197.138,A -85,B 0,C 180,E1 12802.811,E2 12802.811} C_VEL
LIN {X 0,Y 379.135,Z 192.464,A -85,B 0,C 180,E1 12801.342,E2 12801.342} C_VEL
LIN {X 0,Y 374.486,Z 187.041,A -85,B 0,C 180,E1 12799.415,E2 12799.415} C_VEL
LIN {X 0,Y 369.917,Z 181.727,A -85,B 0,C 180,E1 12797.297,E2 12797.297} C_VEL
LIN {X 0,Y 366.386,Z 178.177,A -85,B 0,C 180,E1 12795.349,E2 12795.349} C_VEL
LIN {X 0,Y 365.07,Z 175.338,A -85,B 0,C 180,E1 12793.785,E2 12793.785} C_VEL
LIN {X 0,Y 362.415,Z 171.817,A -85,B 0,C 180,E1 12790.813,E2 12790.813} C_VEL
LIN {X 0,Y 361.539,Z 169.722,A -85,B 0,C 180,E1 12789.23,E2 12789.23} C_VEL
LIN {X 0,Y 358.288,Z 165.266,A -85,B 0,C 180,E1 12781.599,E2 12781.599} C_VEL
LIN {X 0,Y 358.124,Z 164.76,A -85,B 0,C 180,E1 12778.24,E2 12778.24} C_VEL
LIN {X 0,Y 358.461,Z 165.904,A -85,B 0,C 180,E1 12774.558,E2 12774.558} C_VEL
LIN {X 0,Y 361.862,Z 170.271,A -85,B 0,C 180,E1 12767.716,E2 12767.716} C_VEL
LIN {X 0,Y 363.883,Z 174.325,A -85,B 0,C 180,E1 12764.705,E2 12764.705} C_VEL
LIN {X 0,Y 365.355,Z 175.923,A -85,B 0,C 180,E1 12763.297,E2 12763.297} C_VEL
LIN {X 0,Y 367.554,Z 180.021,A -85,B 0,C 180,E1 12760.947,E2 12760.947} C_VEL
LIN {X 0,Y 368.68,Z 181.512,A -85,B 0,C 180,E1 12760.019,E2 12760.019} C_VEL
LIN {X 0,Y 370.775,Z 185.389,A -85,B 0,C 180,E1 12758.152,E2 12758.152} C_VEL
LIN {X 0,Y 371.796,Z 186.936,A -85,B 0,C 180,E1 12757.383,E2 12757.383} C_VEL
LIN {X 0,Y 374.873,Z 192.398,A -85,B 0,C 180,E1 12755.07,E2 12755.07} C_VEL
LIN {X 0,Y 378.025,Z 196.751,A -85,B 0,C 180,E1 12753.576,E2 12753.576} C_VEL
LIN {X 0,Y 383.258,Z 203.733,A -85,B 0,C 180,E1 12751.568,E2 12751.568} C_VEL
LIN {X 0,Y 390.01,Z 212.93,A -85,B 0,C 180,E1 12749.239,E2 12749.239} C_VEL
LIN {X 0,Y 397.398,Z 223.284,A -85,B 0,C 180,E1 12746.952,E2 12746.952} C_VEL
LIN {X 0,Y 407.03,Z 237.813,A -85,B 0,C 180,E1 12744.265,E2 12744.265} C_VEL
LIN {X 0,Y 417.566,Z 255.021,A -85,B 0,C 180,E1 12741.627,E2 12741.627} C_VEL
LIN {X 0,Y 418.029,Z 256.504,A -85,B 0,C 180,E1 12741.498,E2 12741.498} C_VEL
LIN {X 0,Y 418.138,Z 260.305,A -85,B 0,C 180,E1 12741.373,E2 12741.373} C_VEL
LIN {X 0,Y 408.181,Z 489.651,A -85,B 0,C 180,E1 12737.149,E2 12737.149} C_VEL
LIN {X 0,Y 406.536,Z 520.275,A -85,B 0,C 180,E1 12736.538,E2 12736.538} C_VEL
LIN {X 0,Y 404.339,Z 541.867,A -85,B 0,C 180,E1 12735.911,E2 12735.911} C_VEL
LIN {X 0,Y 401.452,Z 562.576,A -85,B 0,C 180,E1 12735.067,E2 12735.067} C_VEL
LIN {X 0,Y 397.987,Z 582.99,A -85,B 0,C 180,E1 12733.998,E2 12733.998} C_VEL
LIN {X 0,Y 394.064,Z 602.071,A -85,B 0,C 180,E1 12732.743,E2 12732.743} C_VEL
LIN {X 0,Y 389.32,Z 622.315,A -85,B 0,C 180,E1 12731.105,E2 12731.105} C_VEL
LIN {X 0,Y 384.486,Z 640.911,A -85,B 0,C 180,E1 12729.281,E2 12729.281} C_VEL
LIN {X 0,Y 379.677,Z 657.799,A -85,B 0,C 180,E1 12727.277,E2 12727.277} C_VEL
LIN {X 0,Y 374.653,Z 674.5,A -85,B 0,C 180,E1 12724.92,E2 12724.92} C_VEL
LIN {X 0,Y 369.924,Z 689.797,A -85,B 0,C 180,E1 12722.354,E2 12722.354} C_VEL
LIN {X 0,Y 365.564,Z 703.619,A -85,B 0,C 180,E1 12719.568,E2 12719.568} C_VEL
LIN {X 0,Y 361.559,Z 716.626,A -85,B 0,C 180,E1 12716.437,E2 12716.437} C_VEL
LIN {X 0,Y 358.304,Z 727.919,A -85,B 0,C 180,E1 12713.17,E2 12713.17} C_VEL
LIN {X 0,Y 355.843,Z 737.254,A -85,B 0,C 180,E1 12709.876,E2 12709.876} C_VEL
LIN {X 0,Y 355.181,Z 739.967,A -85,B 0,C 180,E1 12708.774,E2 12708.774} C_VEL
LIN {X 0,Y 353.587,Z 742.819,A -85,B 0,C 180,E1 12707.629,E2 12707.629} C_VEL
LIN {X 0,Y 346.14,Z 749.583,A -85,B 0,C 180,E1 12704.563,E2 12704.563} C_VEL
LIN {X 0,Y 345.085,Z 751.433,A -85,B 0,C 180,E1 12703.515,E2 12703.515} C_VEL
LIN {X 0,Y 344.391,Z 756.121,A -85,B 0,C 180,E1 12700.032,E2 12700.032} C_VEL
LIN {X 0,Y 344.075,Z 759.6,A -85,B 0,C 180,E1 12696.367,E2 12696.367} C_VEL
LIN {X 0,Y 343.973,Z 761.377,A -85,B 0,C 180,E1 12692.999,E2 12692.999} C_VEL
LIN {X 0,Y 343.956,Z 761.889,A -85,B 0,C 180,E1 12689.334,E2 12689.334} C_VEL
LIN {X 0,Y 343.988,Z 761.094,A -85,B 0,C 180,E1 12686.167,E2 12686.167} C_VEL
LIN {X 0,Y 344.13,Z 758.747,A -85,B 0,C 180,E1 12682.488,E2 12682.488} C_VEL
LIN {X 0,Y 344.531,Z 755.058,A -85,B 0,C 180,E1 12678.958,E2 12678.958} C_VEL
LIN {X 0,Y 345.369,Z 749.769,A -85,B 0,C 180,E1 12675.412,E2 12675.412} C_VEL
LIN {X 0,Y 346.833,Z 742.953,A -85,B 0,C 180,E1 12671.86,E2 12671.86} C_VEL
LIN {X 0,Y 348.929,Z 734.75,A -85,B 0,C 180,E1 12668.483,E2 12668.483} C_VEL
LIN {X 0,Y 351.98,Z 724.259,A -85,B 0,C 180,E1 12664.96,E2 12664.96} C_VEL
LIN {X 0,Y 355.572,Z 712.953,A -85,B 0,C 180,E1 12661.81,E2 12661.81} C_VEL
LIN {X 0,Y 359.726,Z 700.232,A -85,B 0,C 180,E1 12658.871,E2 12658.871} C_VEL
LIN {X 0,Y 364.356,Z 686.22,A -85,B 0,C 180,E1 12656.148,E2 12656.148} C_VEL
LIN {X 0,Y 369.344,Z 670.974,A -85,B 0,C 180,E1 12653.641,E2 12653.641} C_VEL
LIN {X 0,Y 374.544,Z 654.116,A -85,B 0,C 180,E1 12651.343,E2 12651.343} C_VEL
LIN {X 0,Y 379.885,Z 635.732,A -85,B 0,C 180,E1 12649.253,E2 12649.253} C_VEL
LIN {X 0,Y 384.823,Z 617.258,A -85,B 0,C 180,E1 12647.505,E2 12647.505} C_VEL
LIN {X 0,Y 389.373,Z 597.77,A -85,B 0,C 180,E1 12646.005,E2 12646.005} C_VEL
LIN {X 0,Y 393.7,Z 576.373,A -85,B 0,C 180,E1 12644.677,E2 12644.677} C_VEL
LIN {X 0,Y 397.245,Z 555.365,A -85,B 0,C 180,E1 12643.653,E2 12643.653} C_VEL
LIN {X 0,Y 399.907,Z 534.782,A -85,B 0,C 180,E1 12642.906,E2 12642.906} C_VEL
LIN {X 0,Y 402.013,Z 511.426,A -85,B 0,C 180,E1 12642.307,E2 12642.307} C_VEL
LIN {X 0,Y 412.225,Z 286.872,A -85,B 0,C 180,E1 12638.127,E2 12638.127} C_VEL
LIN {X 0,Y 413.406,Z 260.018,A -85,B 0,C 180,E1 12637.596,E2 12637.596} C_VEL
LIN {X 0,Y 403.569,Z 243.718,A -85,B 0,C 180,E1 12635.042,E2 12635.042} C_VEL
LIN {X 0,Y 393.922,Z 229.035,A -85,B 0,C 180,E1 12632.253,E2 12632.253} C_VEL
LIN {X 0,Y 385.739,Z 217.287,A -85,B 0,C 180,E1 12629.59,E2 12629.59} C_VEL
LIN {X 0,Y 378.529,Z 207.562,A -85,B 0,C 180,E1 12626.937,E2 12626.937} C_VEL
LIN {X 0,Y 371.564,Z 198.293,A -85,B 0,C 180,E1 12623.975,E2 12623.975} C_VEL
LIN {X 0,Y 367.87,Z 193.696,A -85,B 0,C 180,E1 12622.198,E2 12622.198} C_VEL
LIN {X 0,Y 365.124,Z 189.899,A -85,B 0,C 180,E1 12620.352,E2 12620.352} C_VEL
LIN {X 0,Y 364.103,Z 187.5,A -85,B 0,C 180,E1 12619.241,E2 12619.241} C_VEL
LIN {X 0,Y 361.514,Z 183.525,A -85,B 0,C 180,E1 12616.717,E2 12616.717} C_VEL
LIN {X 0,Y 360.903,Z 182.177,A -85,B 0,C 180,E1 12615.919,E2 12615.919} C_VEL
LIN {X 0,Y 358.209,Z 178.242,A -85,B 0,C 180,E1 12612.575,E2 12612.575} C_VEL
LIN {X 0,Y 357.545,Z 176.67,A -85,B 0,C 180,E1 12611.289,E2 12611.289} C_VEL
LIN {X 0,Y 354.632,Z 172.709,A -85,B 0,C 180,E1 12604.204,E2 12604.204} C_VEL
LIN {X 0,Y 354.493,Z 172.101,A -85,B 0,C 180,E1 12600.647,E2 12600.647} C_VEL
LIN {X 0,Y 354.898,Z 173.336,A -85,B 0,C 180,E1 12596.77,E2 12596.77} C_VEL
LIN {X 0,Y 358.016,Z 177.229,A -85,B 0,C 180,E1 12590.516,E2 12590.516} C_VEL
LIN {X 0,Y 359.804,Z 180.818,A -85,B 0,C 180,E1 12587.971,E2 12587.971} C_VEL
LIN {X 0,Y 362.944,Z 183.626,A -85,B 0,C 180,E1 12585.97,E2 12585.97} C_VEL
LIN {X 0,Y 367.561,Z 188.722,A -85,B 0,C 180,E1 12583.404,E2 12583.404} C_VEL
LIN {X 0,Y 374.017,Z 196.2,A -85,B 0,C 180,E1 12580.357,E2 12580.357} C_VEL
LIN {X 0,Y 378.865,Z 202.011,A -85,B 0,C 180,E1 12578.358,E2 12578.358} C_VEL
LIN {X 0,Y 383.792,Z 208.1,A -85,B 0,C 180,E1 12576.51,E2 12576.51} C_VEL
LIN {X 0,Y 388.229,Z 213.734,A -85,B 0,C 180,E1 12574.975,E2 12574.975} C_VEL
LIN {X 0,Y 394.707,Z 222.192,A -85,B 0,C 180,E1 12572.914,E2 12572.914} C_VEL
LIN {X 0,Y 404.421,Z 235.81,A -85,B 0,C 180,E1 12570.121,E2 12570.121} C_VEL
LIN {X 0,Y 414.382,Z 250.956,A -85,B 0,C 180,E1 12567.55,E2 12567.55} C_VEL
LIN {X 0,Y 416.593,Z 254.8,A -85,B 0,C 180,E1 12567.002,E2 12567.002} C_VEL
LIN {X 0,Y 405.555,Z 462.707,A -85,B 0,C 180,E1 12562.883,E2 12562.883} C_VEL
LIN {X 0,Y 402.704,Z 513.645,A -85,B 0,C 180,E1 12561.835,E2 12561.835} C_VEL
LIN {X 0,Y 400.184,Z 536.763,A -85,B 0,C 180,E1 12561.158,E2 12561.158} C_VEL
LIN {X 0,Y 396.83,Z 560.405,A -85,B 0,C 180,E1 12560.21,E2 12560.21} C_VEL
LIN {X 0,Y 393.26,Z 581.019,A -85,B 0,C 180,E1 12559.145,E2 12559.145} C_VEL
LIN {X 0,Y 388.911,Z 602.399,A -85,B 0,C 180,E1 12557.766,E2 12557.766} C_VEL
LIN {X 0,Y 384.169,Z 623.319,A -85,B 0,C 180,E1 12556.13,E2 12556.13} C_VEL
LIN {X 0,Y 379.282,Z 642.485,A -85,B 0,C 180,E1 12554.312,E2 12554.312} C_VEL
LIN {X 0,Y 374.023,Z 661.888,A -85,B 0,C 180,E1 12552.142,E2 12552.142} C_VEL
LIN {X 0,Y 369.077,Z 679.23,A -85,B 0,C 180,E1 12549.842,E2 12549.842} C_VEL
LIN {X 0,Y 363.933,Z 696.846,A -85,B 0,C 180,E1 12547.087,E2 12547.087} C_VEL
LIN {X 0,Y 359.343,Z 712.643,A -85,B 0,C 180,E1 12544.197,E2 12544.197} C_VEL
LIN {X 0,Y 355.34,Z 726.543,A -85,B 0,C 180,E1 12541.18,E2 12541.18} C_VEL
LIN {X 0,Y 351.738,Z 739.938,A -85,B 0,C 180,E1 12537.786,E2 12537.786} C_VEL
LIN {X 0,Y 349.065,Z 750.755,A -85,B 0,C 180,E1 12534.54,E2 12534.54} C_VEL
LIN {X 0,Y 346.808,Z 761.275,A -85,B 0,C 180,E1 12530.769,E2 12530.769} C_VEL
LIN {X 0,Y 345.438,Z 769.159,A -85,B 0,C 180,E1 12527.345,E2 12527.345} C_VEL
LIN {X 0,Y 344.53,Z 776.008,A -85,B 0,C 180,E1 12523.595,E2 12523.595} C_VEL
LIN {X 0,Y 344.133,Z 780.574,A -85,B 0,C 180,E1 12520.377,E2 12520.377} C_VEL
LIN {X 0,Y 343.972,Z 784.29,A -85,B 0,C 180,E1 12516.677,E2 12516.677} C_VEL
LIN {X 0,Y 343.939,Z 786.177,A -85,B 0,C 180,E1 12513.5,E2 12513.5} C_VEL
LIN {X 0,Y 343.948,Z 786.978,A -85,B 0,C 180,E1 12510,E2 12510} C_VEL
LIN {X 0,Y 343.939,Z 786.177,A -85,B 0,C 180,E1 12506.5,E2 12506.5} C_VEL
LIN {X 0,Y 343.972,Z 784.289,A -85,B 0,C 180,E1 12503.323,E2 12503.323} C_VEL
LIN {X 0,Y 344.133,Z 780.574,A -85,B 0,C 180,E1 12499.623,E2 12499.623} C_VEL
LIN {X 0,Y 344.53,Z 776.008,A -85,B 0,C 180,E1 12496.405,E2 12496.405} C_VEL
LIN {X 0,Y 345.439,Z 769.155,A -85,B 0,C 180,E1 12492.655,E2 12492.655} C_VEL
LIN {X 0,Y 346.808,Z 761.272,A -85,B 0,C 180,E1 12489.231,E2 12489.231} C_VEL
LIN {X 0,Y 349.066,Z 750.753,A -85,B 0,C 180,E1 12485.46,E2 12485.46} C_VEL
LIN {X 0,Y 351.738,Z 739.933,A -85,B 0,C 180,E1 12482.214,E2 12482.214} C_VEL
LIN {X 0,Y 355.369,Z 726.424,A -85,B 0,C 180,E1 12478.795,E2 12478.795} C_VEL
LIN {X 0,Y 359.499,Z 712.063,A -85,B 0,C 180,E1 12475.693,E2 12475.693} C_VEL
LIN {X 0,Y 364.071,Z 696.341,A -85,B 0,C 180,E1 12472.83,E2 12472.83} C_VEL
LIN {X 0,Y 369.387,Z 678.062,A -85,B 0,C 180,E1 12469.998,E2 12469.998} C_VEL
LIN {X 0,Y 374.574,Z 659.963,A -85,B 0,C 180,E1 12467.625,E2 12467.625} C_VEL
LIN {X 0,Y 379.663,Z 640.91,A -85,B 0,C 180,E1 12465.533,E2 12465.533} C_VEL
LIN {X 0,Y 384.775,Z 620.522,A -85,B 0,C 180,E1 12463.641,E2 12463.641} C_VEL
LIN {X 0,Y 389.349,Z 600.261,A -85,B 0,C 180,E1 12462.086,E2 12462.086} C_VEL
LIN {X 0,Y 393.806,Z 577.794,A -85,B 0,C 180,E1 12460.682,E2 12460.682} C_VEL
LIN {X 0,Y 397.624,Z 555.453,A -85,B 0,C 180,E1 12459.569,E2 12459.569} C_VEL
LIN {X 0,Y 400.549,Z 533.548,A -85,B 0,C 180,E1 12458.742,E2 12458.742} C_VEL
LIN {X 0,Y 402.976,Z 509.197,A -85,B 0,C 180,E1 12458.071,E2 12458.071} C_VEL
LIN {X 0,Y 412.979,Z 320.624,A -85,B 0,C 180,E1 12454.3,E2 12454.3} C_VEL
LIN {X 0,Y 416.476,Z 254.395,A -85,B 0,C 180,E1 12452.982,E2 12452.982} C_VEL
LIN {X 0,Y 406.333,Z 238.689,A -85,B 0,C 180,E1 12450.416,E2 12450.416} C_VEL
LIN {X 0,Y 396.8,Z 225.086,A -85,B 0,C 180,E1 12447.744,E2 12447.744} C_VEL
LIN {X 0,Y 388.751,Z 214.415,A -85,B 0,C 180,E1 12445.233,E2 12445.233} C_VEL
LIN {X 0,Y 384.567,Z 209.09,A -85,B 0,C 180,E1 12443.806,E2 12443.806} C_VEL
LIN {X 0,Y 380.668,Z 204.271,A -85,B 0,C 180,E1 12442.386,E2 12442.386} C_VEL
LIN {X 0,Y 376.713,Z 199.436,A -85,B 0,C 180,E1 12440.834,E2 12440.834} C_VEL
LIN {X 0,Y 372.501,Z 194.422,A -85,B 0,C 180,E1 12439.034,E2 12439.034} C_VEL
LIN {X 0,Y 367.42,Z 188.609,A -85,B 0,C 180,E1 12436.603,E2 12436.603} C_VEL
LIN {X 0,Y 362.921,Z 183.596,A -85,B 0,C 180,E1 12434.112,E2 12434.112} C_VEL
LIN {X 0,Y 358.853,Z 179.548,A -85,B 0,C 180,E1 12431.247,E2 12431.247} C_VEL
LIN {X 0,Y 357.703,Z 176.735,A -85,B 0,C 180,E1 12429.168,E2 12429.168} C_VEL
LIN {X 0,Y 354.526,Z 172.284,A -85,B 0,C 180,E1 12421.454,E2 12421.454} C_VEL
LIN {X 0,Y 354.376,Z 171.829,A -85,B 0,C 180,E1 12418.221,E2 12418.221} C_VEL
LIN {X 0,Y 354.704,Z 173.009,A -85,B 0,C 180,E1 12414.5,E2 12414.5} C_VEL
LIN {X 0,Y 357.916,Z 177.159,A -85,B 0,C 180,E1 12407.882,E2 12407.882} C_VEL
LIN {X 0,Y 359.866,Z 181.183,A -85,B 0,C 180,E1 12404.86,E2 12404.86} C_VEL
LIN {X 0,Y 361.285,Z 182.828,A -85,B 0,C 180,E1 12403.438,E2 12403.438} C_VEL
LIN {X 0,Y 363.678,Z 187.082,A -85,B 0,C 180,E1 12400.903,E2 12400.903} C_VEL
LIN {X 0,Y 364.536,Z 188.478,A -85,B 0,C 180,E1 12400.116,E2 12400.116} C_VEL
LIN {X 0,Y 367.02,Z 192.558,A -85,B 0,C 180,E1 12398.085,E2 12398.085} C_VEL
LIN {X 0,Y 371.59,Z 198.334,A -85,B 0,C 180,E1 12395.858,E2 12395.858} C_VEL
LIN {X 0,Y 380.065,Z 209.525,A -85,B 0,C 180,E1 12392.333,E2 12392.333} C_VEL
LIN {X 0,Y 387.524,Z 219.983,A -85,B 0,C 180,E1 12389.665,E2 12389.665} C_VEL
LIN {X 0,Y 395.348,Z 231.101,A -85,B 0,C 180,E1 12387.19,E2 12387.19} C_VEL
LIN {X 0,Y 404.872,Z 245.978,A -85,B 0,C 180,E1 12384.481,E2 12384.481} C_VEL
LIN {X 0,Y 413.471,Z 260.264,A -85,B 0,C 180,E1 12382.274,E2 12382.274} C_VEL
LIN {X 0,Y 403.008,Z 489.962,A -85,B 0,C 180,E1 12378.01,E2 12378.01} C_VEL
LIN {X 0,Y 401.3,Z 520.35,A -85,B 0,C 180,E1 12377.398,E2 12377.398} C_VEL
LIN {X 0,Y 399.008,Z 542.049,A -85,B 0,C 180,E1 12376.766,E2 12376.766} C_VEL
LIN {X 0,Y 395.882,Z 563.534,A -85,B 0,C 180,E1 12375.881,E2 12375.881} C_VEL
LIN {X 0,Y 392.056,Z 584.849,A -85,B 0,C 180,E1 12374.738,E2 12374.738} C_VEL
LIN {X 0,Y 388.011,Z 603.729,A -85,B 0,C 180,E1 12373.473,E2 12373.473} C_VEL
LIN {X 0,Y 383.303,Z 622.873,A -85,B 0,C 180,E1 12371.895,E2 12371.895} C_VEL
LIN {X 0,Y 378.482,Z 640.7,A -85,B 0,C 180,E1 12370.133,E2 12370.133} C_VEL
LIN {X 0,Y 373.312,Z 658.086,A -85,B 0,C 180,E1 12368.053,E2 12368.053} C_VEL
LIN {X 0,Y 368.123,Z 674.588,A -85,B 0,C 180,E1 12365.697,E2 12365.697} C_VEL
LIN {X 0,Y 363.338,Z 689.347,A -85,B 0,C 180,E1 12363.203,E2 12363.203} C_VEL
LIN {X 0,Y 358.613,Z 703.567,A -85,B 0,C 180,E1 12360.307,E2 12360.307} C_VEL
LIN {X 0,Y 354.441,Z 716.372,A -85,B 0,C 180,E1 12357.192,E2 12357.192} C_VEL
LIN {X 0,Y 351.099,Z 727.267,A -85,B 0,C 180,E1 12354.031,E2 12354.031} C_VEL
LIN {X 0,Y 348.388,Z 736.711,A -85,B 0,C 180,E1 12350.671,E2 12350.671} C_VEL
LIN {X 0,Y 346.302,Z 745.198,A -85,B 0,C 180,E1 12346.954,E2 12346.954} C_VEL
LIN {X 0,Y 345.085,Z 751.433,A -85,B 0,C 180,E1 12343.515,E2 12343.515} C_VEL
LIN {X 0,Y 343.79,Z 753.403,A -85,B 0,C 180,E1 12342.285,E2 12342.285} C_VEL
LIN {X 0,Y 336.895,Z 757.89,A -85,B 0,C 180,E1 12338.874,E2 12338.874} C_VEL
LIN {X 0,Y 336.167,Z 758.822,A -85,B 0,C 180,E1 12337.849,E2 12337.849} C_VEL
LIN {X 0,Y 336.002,Z 761.286,A -85,B 0,C 180,E1 12334.095,E2 12334.095} C_VEL
LIN {X 0,Y 335.961,Z 762.167,A -85,B 0,C 180,E1 12330.682,E2 12330.682} C_VEL
LIN {X 0,Y 335.978,Z 761.769,A -85,B 0,C 180,E1 12327.1,E2 12327.1} C_VEL
LIN {X 0,Y 336.074,Z 760.079,A -85,B 0,C 180,E1 12323.68,E2 12323.68} C_VEL
LIN {X 0,Y 336.401,Z 756.726,A -85,B 0,C 180,E1 12319.901,E2 12319.901} C_VEL
LIN {X 0,Y 337.142,Z 752.059,A -85,B 0,C 180,E1 12316.276,E2 12316.276} C_VEL
LIN {X 0,Y 338.507,Z 745.55,A -85,B 0,C 180,E1 12312.565,E2 12312.565} C_VEL
LIN {X 0,Y 340.811,Z 736.834,A -85,B 0,C 180,E1 12308.668,E2 12308.668} C_VEL
LIN {X 0,Y 343.808,Z 727.054,A -85,B 0,C 180,E1 12305.143,E2 12305.143} C_VEL
LIN {X 0,Y 347.496,Z 715.818,A -85,B 0,C 180,E1 12301.844,E2 12301.844} C_VEL
LIN {X 0,Y 351.967,Z 702.834,A -85,B 0,C 180,E1 12298.678,E2 12298.678} C_VEL
LIN {X 0,Y 356.709,Z 689.311,A -85,B 0,C 180,E1 12295.904,E2 12295.904} C_VEL
LIN {X 0,Y 361.798,Z 674.352,A -85,B 0,C 180,E1 12293.351,E2 12293.351} C_VEL
LIN {X 0,Y 367.496,Z 656.939,A -85,B 0,C 180,E1 12290.862,E2 12290.862} C_VEL
LIN {X 0,Y 372.768,Z 639.941,A -85,B 0,C 180,E1 12288.831,E2 12288.831} C_VEL
LIN {X 0,Y 377.734,Z 622.203,A -85,B 0,C 180,E1 12287.082,E2 12287.082} C_VEL
LIN {X 0,Y 382.745,Z 602.384,A -85,B 0,C 180,E1 12285.461,E2 12285.461} C_VEL
LIN {X 0,Y 386.941,Z 583.403,A -85,B 0,C 180,E1 12284.198,E2 12284.198} C_VEL
LIN {X 0,Y 390.748,Z 562.581,A -85,B 0,C 180,E1 12283.095,E2 12283.095} C_VEL
LIN {X 0,Y 393.958,Z 541.023,A -85,B 0,C 180,E1 12282.221,E2 12282.221} C_VEL
LIN {X 0,Y 396.283,Z 519.659,A -85,B 0,C 180,E1 12281.603,E2 12281.603} C_VEL
LIN {X 0,Y 398.078,Z 488.141,A -85,B 0,C 180,E1 12280.97,E2 12280.97} C_VEL
LIN {X 0,Y 408.765,Z 264.154,A -85,B 0,C 180,E1 12276.78,E2 12276.78} C_VEL
LIN {X 0,Y 399.483,Z 248.757,A -85,B 0,C 180,E1 12274.274,E2 12274.274} C_VEL
LIN {X 0,Y 390.727,Z 235.142,A -85,B 0,C 180,E1 12271.641,E2 12271.641} C_VEL
LIN {X 0,Y 382.714,Z 223.532,A -85,B 0,C 180,E1 12268.941,E2 12268.941} C_VEL
LIN {X 0,Y 376.235,Z 214.618,A -85,B 0,C 180,E1 12266.475,E2 12266.475} C_VEL
LIN {X 0,Y 369.498,Z 205.535,A -85,B 0,C 180,E1 12263.524,E2 12263.524} C_VEL
LIN {X 0,Y 365.769,Z 200.618,A -85,B 0,C 180,E1 12261.656,E2 12261.656} C_VEL
LIN {X 0,Y 361.654,Z 195.519,A -85,B 0,C 180,E1 12259.334,E2 12259.334} C_VEL
LIN {X 0,Y 357.318,Z 189.904,A -85,B 0,C 180,E1 12256.308,E2 12256.308} C_VEL
LIN {X 0,Y 356.525,Z 188.753,A -85,B 0,C 180,E1 12255.452,E2 12255.452} C_VEL
LIN {X 0,Y 354.186,Z 184.854,A -85,B 0,C 180,E1 12252.224,E2 12252.224} C_VEL
LIN {X 0,Y 353.467,Z 183.481,A -85,B 0,C 180,E1 12250.925,E2 12250.925} C_VEL
LIN {X 0,Y 350.855,Z 179.737,A -85,B 0,C 180,E1 12244.086,E2 12244.086} C_VEL
LIN {X 0,Y 350.742,Z 179.169,A -85,B 0,C 180,E1 12240.654,E2 12240.654} C_VEL
LIN {X 0,Y 351.144,Z 180.432,A -85,B 0,C 180,E1 12236.736,E2 12236.736} C_VEL
LIN {X 0,Y 352.984,Z 182.858,A -85,B 0,C 180,E1 12232.841,E2 12232.841} C_VEL
LIN {X 0,Y 355.376,Z 184.829,A -85,B 0,C 180,E1 12230.608,E2 12230.608} C_VEL
LIN {X 0,Y 360.219,Z 190.091,A -85,B 0,C 180,E1 12227.007,E2 12227.007} C_VEL
LIN {X 0,Y 361.684,Z 191.703,A -85,B 0,C 180,E1 12226.084,E2 12226.084} C_VEL
LIN {X 0,Y 366.845,Z 197.486,A -85,B 0,C 180,E1 12223.208,E2 12223.208} C_VEL
LIN {X 0,Y 372.106,Z 203.664,A -85,B 0,C 180,E1 12220.701,E2 12220.701} C_VEL
LIN {X 0,Y 376.873,Z 209.492,A -85,B 0,C 180,E1 12218.687,E2 12218.687} C_VEL
LIN {X 0,Y 381.822,Z 215.709,A -85,B 0,C 180,E1 12216.79,E2 12216.79} C_VEL
LIN {X 0,Y 388.033,Z 223.664,A -85,B 0,C 180,E1 12214.635,E2 12214.635} C_VEL
LIN {X 0,Y 397.88,Z 237.307,A -85,B 0,C 180,E1 12211.584,E2 12211.584} C_VEL
LIN {X 0,Y 407.701,Z 252.091,A -85,B 0,C 180,E1 12208.879,E2 12208.879} C_VEL
LIN {X 0,Y 411.747,Z 258.892,A -85,B 0,C 180,E1 12207.83,E2 12207.83} C_VEL
LIN {X 0,Y 400.338,Z 465.82,A -85,B 0,C 180,E1 12203.707,E2 12203.707} C_VEL
LIN {X 0,Y 397.534,Z 513.775,A -85,B 0,C 180,E1 12202.711,E2 12202.711} C_VEL
LIN {X 0,Y 394.945,Z 536.812,A -85,B 0,C 180,E1 12202.035,E2 12202.035} C_VEL
LIN {X 0,Y 391.414,Z 560.782,A -85,B 0,C 180,E1 12201.068,E2 12201.068} C_VEL
LIN {X 0,Y 387.456,Z 582.785,A -85,B 0,C 180,E1 12199.917,E2 12199.917} C_VEL
LIN {X 0,Y 382.949,Z 603.77,A -85,B 0,C 180,E1 12198.531,E2 12198.531} C_VEL
LIN {X 0,Y 378.029,Z 624.407,A -85,B 0,C 180,E1 12196.885,E2 12196.885} C_VEL
LIN {X 0,Y 372.965,Z 643.453,A -85,B 0,C 180,E1 12195.05,E2 12195.05} C_VEL
LIN {X 0,Y 367.116,Z 663.91,A -85,B 0,C 180,E1 12192.699,E2 12192.699} C_VEL
LIN {X 0,Y 361.853,Z 681.626,A -85,B 0,C 180,E1 12190.283,E2 12190.283} C_VEL
LIN {X 0,Y 356.672,Z 698.336,A -85,B 0,C 180,E1 12187.568,E2 12187.568} C_VEL
LIN {X 0,Y 351.643,Z 714.666,A -85,B 0,C 180,E1 12184.454,E2 12184.454} C_VEL
LIN {X 0,Y 347.399,Z 728.836,A -85,B 0,C 180,E1 12181.262,E2 12181.262} C_VEL
LIN {X 0,Y 343.769,Z 741.594,A -85,B 0,C 180,E1 12177.849,E2 12177.849} C_VEL
LIN {X 0,Y 340.853,Z 753.028,A -85,B 0,C 180,E1 12174.247,E2 12174.247} C_VEL
LIN {X 0,Y 338.757,Z 762.38,A -85,B 0,C 180,E1 12170.669,E2 12170.669} C_VEL
LIN {X 0,Y 337.252,Z 770.809,A -85,B 0,C 180,E1 12166.744,E2 12166.744} C_VEL
LIN {X 0,Y 336.47,Z 776.76,A -85,B 0,C 180,E1 12163.227,E2 12163.227} C_VEL
LIN {X 0,Y 336.067,Z 781.635,A -85,B 0,C 180,E1 12159.418,E2 12159.418} C_VEL
LIN {X 0,Y 335.959,Z 784.472,A -85,B 0,C 180,E1 12156.15,E2 12156.15} C_VEL
LIN {X 0,Y 335.944,Z 786.314,A -85,B 0,C 180,E1 12152.559,E2 12152.559} C_VEL
LIN {X 0,Y 335.95,Z 786.552,A -85,B 0,C 180,E1 12148.977,E2 12148.977} C_VEL
LIN {X 0,Y 335.942,Z 785.666,A -85,B 0,C 180,E1 12145.904,E2 12145.904} C_VEL
LIN {X 0,Y 336.006,Z 783.154,A -85,B 0,C 180,E1 12142.133,E2 12142.133} C_VEL
LIN {X 0,Y 336.226,Z 779.388,A -85,B 0,C 180,E1 12138.681,E2 12138.681} C_VEL
LIN {X 0,Y 336.8,Z 774.052,A -85,B 0,C 180,E1 12135.033,E2 12135.033} C_VEL
LIN {X 0,Y 337.888,Z 766.963,A -85,B 0,C 180,E1 12131.363,E2 12131.363} C_VEL
LIN {X 0,Y 339.72,Z 757.922,A -85,B 0,C 180,E1 12127.541,E2 12127.541} C_VEL
LIN {X 0,Y 342.025,Z 748.24,A -85,B 0,C 180,E1 12124.179,E2 12124.179} C_VEL
LIN {X 0,Y 345.39,Z 735.749,A -85,B 0,C 180,E1 12120.52,E2 12120.52} C_VEL
LIN {X 0,Y 349.272,Z 722.501,A -85,B 0,C 180,E1 12117.246,E2 12117.246} C_VEL
LIN {X 0,Y 353.719,Z 707.852,A -85,B 0,C 180,E1 12114.189,E2 12114.189} C_VEL
LIN {X 0,Y 358.727,Z 691.706,A -85,B 0,C 180,E1 12111.299,E2 12111.299} C_VEL
LIN {X 0,Y 363.888,Z 674.732,A -85,B 0,C 180,E1 12108.743,E2 12108.743} C_VEL
LIN {X 0,Y 369.683,Z 655.007,A -85,B 0,C 180,E1 12106.231,E2 12106.231} C_VEL
LIN {X 0,Y 375.017,Z 635.86,A -85,B 0,C 180,E1 12104.178,E2 12104.178} C_VEL
LIN {X 0,Y 379.98,Z 616.226,A -85,B 0,C 180,E1 12102.433,E2 12102.433} C_VEL
LIN {X 0,Y 384.825,Z 595.334,A -85,B 0,C 180,E1 12100.882,E2 12100.882} C_VEL
LIN {X 0,Y 388.938,Z 574.718,A -85,B 0,C 180,E1 12099.642,E2 12099.642} C_VEL
LIN {X 0,Y 392.877,Z 551.444,A -85,B 0,C 180,E1 12098.53,E2 12098.53} C_VEL
LIN {X 0,Y 395.616,Z 531.299,A -85,B 0,C 180,E1 12097.792,E2 12097.792} C_VEL
LIN {X 0,Y 397.967,Z 507.101,A -85,B 0,C 180,E1 12097.144,E2 12097.144} C_VEL
LIN {X 0,Y 408.715,Z 311.819,A -85,B 0,C 180,E1 12093.224,E2 12093.224} C_VEL
LIN {X 0,Y 411.581,Z 258.416,A -85,B 0,C 180,E1 12092.142,E2 12092.142} C_VEL
LIN {X 0,Y 402.604,Z 244.387,A -85,B 0,C 180,E1 12089.781,E2 12089.781} C_VEL
LIN {X 0,Y 393.809,Z 231.656,A -85,B 0,C 180,E1 12087.235,E2 12087.235} C_VEL
LIN {X 0,Y 386.118,Z 221.279,A -85,B 0,C 180,E1 12084.762,E2 12084.762} C_VEL
LIN {X 0,Y 379.678,Z 212.851,A -85,B 0,C 180,E1 12082.448,E2 12082.448} C_VEL
LIN {X 0,Y 374.15,Z 206.2,A -85,B 0,C 180,E1 12080.247,E2 12080.247} C_VEL
LIN {X 0,Y 370.372,Z 201.64,A -85,B 0,C 180,E1 12078.575,E2 12078.575} C_VEL
LIN {X 0,Y 365.701,Z 196.163,A -85,B 0,C 180,E1 12076.274,E2 12076.274} C_VEL
LIN {X 0,Y 361.181,Z 190.94,A -85,B 0,C 180,E1 12073.691,E2 12073.691} C_VEL
LIN {X 0,Y 355.567,Z 185.114,A -85,B 0,C 180,E1 12069.713,E2 12069.713} C_VEL
LIN {X 0,Y 354.111,Z 183.73,A -85,B 0,C 180,E1 12068.443,E2 12068.443} C_VEL
LIN {X 0,Y 351.654,Z 181.442,A -85,B 0,C 180,E1 12065.384,E2 12065.384} C_VEL
LIN {X 0,Y 350.698,Z 179.112,A -85,B 0,C 180,E1 12060.653,E2 12060.653} C_VEL
LIN {X 0,Y 350.664,Z 178.975,A -85,B 0,C 180,E1 12057.385,E2 12057.385} C_VEL
LIN {X 0,Y 351.262,Z 180.809,A -85,B 0,C 180,E1 12053.134,E2 12053.134} C_VEL
LIN {X 0,Y 354.018,Z 184.23,A -85,B 0,C 180,E1 12047.936,E2 12047.936} C_VEL
LIN {X 0,Y 356.155,Z 188.386,A -85,B 0,C 180,E1 12044.699,E2 12044.699} C_VEL
LIN {X 0,Y 357.262,Z 189.749,A -85,B 0,C 180,E1 12043.58,E2 12043.58} C_VEL
LIN {X 0,Y 360.677,Z 194.419,A -85,B 0,C 180,E1 12041.074,E2 12041.074} C_VEL
LIN {X 0,Y 362.051,Z 196.241,A -85,B 0,C 180,E1 12040.226,E2 12040.226} C_VEL
LIN {X 0,Y 366.11,Z 201.246,A -85,B 0,C 180,E1 12037.986,E2 12037.986} C_VEL
LIN {X 0,Y 371.185,Z 207.893,A -85,B 0,C 180,E1 12035.534,E2 12035.534} C_VEL
LIN {X 0,Y 377.916,Z 216.847,A -85,B 0,C 180,E1 12032.718,E2 12032.718} C_VEL
LIN {X 0,Y 385.056,Z 227.033,A -85,B 0,C 180,E1 12030.095,E2 12030.095} C_VEL
LIN {X 0,Y 392.538,Z 237.882,A -85,B 0,C 180,E1 12027.662,E2 12027.662} C_VEL
LIN {X 0,Y 401.569,Z 252.205,A -85,B 0,C 180,E1 12025.019,E2 12025.019} C_VEL
LIN {X 0,Y 408.697,Z 264.332,A -85,B 0,C 180,E1 12023.117,E2 12023.117} C_VEL
LIN {X 0,Y 397.805,Z 493.019,A -85,B 0,C 180,E1 12018.843,E2 12018.843} C_VEL
LIN {X 0,Y 395.993,Z 522.063,A -85,B 0,C 180,E1 12018.24,E2 12018.24} C_VEL
LIN {X 0,Y 393.551,Z 543.91,A -85,B 0,C 180,E1 12017.584,E2 12017.584} C_VEL
LIN {X 0,Y 390.394,Z 564.481,A -85,B 0,C 180,E1 12016.718,E2 12016.718} C_VEL
LIN {X 0,Y 386.284,Z 586.265,A -85,B 0,C 180,E1 12015.527,E2 12015.527} C_VEL
LIN {X 0,Y 381.796,Z 606.326,A -85,B 0,C 180,E1 12014.154,E2 12014.154} C_VEL
LIN {X 0,Y 376.927,Z 625.019,A -85,B 0,C 180,E1 12012.564,E2 12012.564} C_VEL
LIN {X 0,Y 371.333,Z 644.449,A -85,B 0,C 180,E1 12010.56,E2 12010.56} C_VEL
LIN {X 0,Y 366.006,Z 661.653,A -85,B 0,C 180,E1 12008.424,E2 12008.424} C_VEL
LIN {X 0,Y 360.606,Z 677.798,A -85,B 0,C 180,E1 12006.001,E2 12006.001} C_VEL
LIN {X 0,Y 355.362,Z 693.025,A -85,B 0,C 180,E1 12003.274,E2 12003.274} C_VEL
LIN {X 0,Y 350.586,Z 706.868,A -85,B 0,C 180,E1 12000.317,E2 12000.317} C_VEL
LIN {X 0,Y 346.362,Z 719.172,A -85,B 0,C 180,E1 11997.135,E2 11997.135} C_VEL
LIN {X 0,Y 342.759,Z 730.297,A -85,B 0,C 180,E1 11993.656,E2 11993.656} C_VEL
LIN {X 0,Y 340.052,Z 739.585,A -85,B 0,C 180,E1 11990.121,E2 11990.121} C_VEL
LIN {X 0,Y 338.127,Z 747.198,A -85,B 0,C 180,E1 11986.491,E2 11986.491} C_VEL
LIN {X 0,Y 336.89,Z 753.373,A -85,B 0,C 180,E1 11982.687,E2 11982.687} C_VEL
LIN {X 0,Y 336.285,Z 757.757,A -85,B 0,C 180,E1 11979.066,E2 11979.066} C_VEL
LIN {X 0,Y 336.167,Z 758.822,A -85,B 0,C 180,E1 11977.849,E2 11977.849} C_VEL
LIN {X 0,Y 335.094,Z 759.937,A -85,B 0,C 180,E1 11976.551,E2 11976.551} C_VEL
LIN {X 0,Y 330.561,Z 761.56,A -85,B 0,C 180,E1 11974.182,E2 11974.182} C_VEL
LIN {X 0,Y 328.185,Z 762.216,A -85,B 0,C 180,E1 11972.477,E2 11972.477} C_VEL
LIN {X 0,Y 327.972,Z 762.313,A -85,B 0,C 180,E1 11971.892,E2 11971.892} C_VEL
LIN {X 0,Y 327.974,Z 762.384,A -85,B 0,C 180,E1 11968.603,E2 11968.603} C_VEL
LIN {X 0,Y 328.03,Z 761.228,A -85,B 0,C 180,E1 11964.929,E2 11964.929} C_VEL
LIN {X 0,Y 328.247,Z 758.738,A -85,B 0,C 180,E1 11961.416,E2 11961.416} C_VEL
LIN {X 0,Y 328.873,Z 754.353,A -85,B 0,C 180,E1 11957.403,E2 11957.403} C_VEL
LIN {X 0,Y 330.063,Z 748.66,A -85,B 0,C 180,E1 11953.637,E2 11953.637} C_VEL
LIN {X 0,Y 331.98,Z 741.27,A -85,B 0,C 180,E1 11949.92,E2 11949.92} C_VEL
LIN {X 0,Y 334.95,Z 731.652,A -85,B 0,C 180,E1 11946.049,E2 11946.049} C_VEL
LIN {X 0,Y 338.589,Z 721.056,A -85,B 0,C 180,E1 11942.57,E2 11942.57} C_VEL
LIN {X 0,Y 342.917,Z 708.924,A -85,B 0,C 180,E1 11939.32,E2 11939.32} C_VEL
LIN {X 0,Y 347.84,Z 695.459,A -85,B 0,C 180,E1 11936.306,E2 11936.306} C_VEL
LIN {X 0,Y 353.237,Z 680.673,A -85,B 0,C 180,E1 11933.53,E2 11933.53} C_VEL
LIN {X 0,Y 358.577,Z 665.327,A -85,B 0,C 180,E1 11931.143,E2 11931.143} C_VEL
LIN {X 0,Y 364.455,Z 647.537,A -85,B 0,C 180,E1 11928.822,E2 11928.822} C_VEL
LIN {X 0,Y 370.058,Z 629.289,A -85,B 0,C 180,E1 11926.846,E2 11926.846} C_VEL
LIN {X 0,Y 375.197,Z 610.44,A -85,B 0,C 180,E1 11925.183,E2 11925.183} C_VEL
LIN {X 0,Y 380.211,Z 589.618,A -85,B 0,C 180,E1 11923.684,E2 11923.684} C_VEL
LIN {X 0,Y 384.327,Z 569.657,A -85,B 0,C 180,E1 11922.532,E2 11922.532} C_VEL
LIN {X 0,Y 387.75,Z 548.738,A -85,B 0,C 180,E1 11921.602,E2 11921.602} C_VEL
LIN {X 0,Y 390.548,Z 526.765,A -85,B 0,C 180,E1 11920.878,E2 11920.878} C_VEL
LIN {X 0,Y 392.331,Z 504.593,A -85,B 0,C 180,E1 11920.368,E2 11920.368} C_VEL
LIN {X 0,Y 403.5,Z 279.162,A -85,B 0,C 180,E1 11916.126,E2 11916.126} C_VEL
LIN {X 0,Y 403.998,Z 267.962,A -85,B 0,C 180,E1 11915.891,E2 11915.891} C_VEL
LIN {X 0,Y 393.946,Z 251.168,A -85,B 0,C 180,E1 11913.028,E2 11913.028} C_VEL
LIN {X 0,Y 384.827,Z 237.08,A -85,B 0,C 180,E1 11910.096,E2 11910.096} C_VEL
LIN {X 0,Y 376.892,Z 225.752,A -85,B 0,C 180,E1 11907.192,E2 11907.192} C_VEL
LIN {X 0,Y 372.85,Z 220.175,A -85,B 0,C 180,E1 11905.536,E2 11905.536} C_VEL
LIN {X 0,Y 367.146,Z 212.433,A -85,B 0,C 180,E1 11902.92,E2 11902.92} C_VEL
LIN {X 0,Y 363.119,Z 207.113,A -85,B 0,C 180,E1 11900.806,E2 11900.806} C_VEL
LIN {X 0,Y 359.155,Z 202.018,A -85,B 0,C 180,E1 11898.42,E2 11898.42} C_VEL
LIN {X 0,Y 355.573,Z 197.155,A -85,B 0,C 180,E1 11895.829,E2 11895.829} C_VEL
LIN {X 0,Y 351.507,Z 192.36,A -85,B 0,C 180,E1 11892.068,E2 11892.068} C_VEL
LIN {X 0,Y 350.524,Z 190.906,A -85,B 0,C 180,E1 11890.852,E2 11890.852} C_VEL
LIN {X 0,Y 347.47,Z 186.961,A -85,B 0,C 180,E1 11883.96,E2 11883.96} C_VEL
LIN {X 0,Y 347.649,Z 186.583,A -85,B 0,C 180,E1 11880.495,E2 11880.495} C_VEL
LIN {X 0,Y 349.143,Z 188.298,A -85,B 0,C 180,E1 11876.552,E2 11876.552} C_VEL
LIN {X 0,Y 354.025,Z 192.505,A -85,B 0,C 180,E1 11870.9,E2 11870.9} C_VEL
LIN {X 0,Y 358.754,Z 197.788,A -85,B 0,C 180,E1 11867.281,E2 11867.281} C_VEL
LIN {X 0,Y 360.189,Z 199.407,A -85,B 0,C 180,E1 11866.352,E2 11866.352} C_VEL
LIN {X 0,Y 365.19,Z 205.131,A -85,B 0,C 180,E1 11863.498,E2 11863.498} C_VEL
LIN {X 0,Y 370.369,Z 211.34,A -85,B 0,C 180,E1 11860.975,E2 11860.975} C_VEL
LIN {X 0,Y 374.808,Z 216.847,A -85,B 0,C 180,E1 11859.056,E2 11859.056} C_VEL
LIN {X 0,Y 381.684,Z 225.502,A -85,B 0,C 180,E1 11856.413,E2 11856.413} C_VEL
LIN {X 0,Y 390.196,Z 237.277,A -85,B 0,C 180,E1 11853.521,E2 11853.521} C_VEL
LIN {X 0,Y 398.78,Z 249.77,A -85,B 0,C 180,E1 11850.936,E2 11850.936} C_VEL
LIN {X 0,Y 407.003,Z 262.661,A -85,B 0,C 180,E1 11848.685,E2 11848.685} C_VEL
LIN {X 0,Y 395.287,Z 467.525,A -85,B 0,C 180,E1 11844.581,E2 11844.581} C_VEL
LIN {X 0,Y 392.448,Z 514.039,A -85,B 0,C 180,E1 11843.607,E2 11843.607} C_VEL
LIN {X 0,Y 389.793,Z 536.931,A -85,B 0,C 180,E1 11842.932,E2 11842.932} C_VEL
LIN {X 0,Y 386.093,Z 561.152,A -85,B 0,C 180,E1 11841.951,E2 11841.951} C_VEL
LIN {X 0,Y 381.966,Z 583.251,A -85,B 0,C 180,E1 11840.787,E2 11840.787} C_VEL
LIN {X 0,Y 377.294,Z 604.129,A -85,B 0,C 180,E1 11839.396,E2 11839.396} C_VEL
LIN {X 0,Y 371.957,Z 625.503,A -85,B 0,C 180,E1 11837.664,E2 11837.664} C_VEL
LIN {X 0,Y 366.922,Z 643.679,A -85,B 0,C 180,E1 11835.891,E2 11835.891} C_VEL
LIN {X 0,Y 361.029,Z 663.442,A -85,B 0,C 180,E1 11833.597,E2 11833.597} C_VEL
LIN {X 0,Y 355.493,Z 681.177,A -85,B 0,C 180,E1 11831.157,E2 11831.157} C_VEL
LIN {X 0,Y 350.049,Z 697.922,A -85,B 0,C 180,E1 11828.406,E2 11828.406} C_VEL
LIN {X 0,Y 345.012,Z 713.461,A -85,B 0,C 180,E1 11825.422,E2 11825.422} C_VEL
LIN {X 0,Y 340.595,Z 727.287,A -85,B 0,C 180,E1 11822.279,E2 11822.279} C_VEL
LIN {X 0,Y 336.616,Z 740.406,A -85,B 0,C 180,E1 11818.762,E2 11818.762} C_VEL
LIN {X 0,Y 333.514,Z 751.654,A -85,B 0,C 180,E1 11815.195,E2 11815.195} C_VEL
LIN {X 0,Y 331.127,Z 761.444,A -85,B 0,C 180,E1 11811.43,E2 11811.43} C_VEL
LIN {X 0,Y 329.533,Z 769.585,A -85,B 0,C 180,E1 11807.662,E2 11807.662} C_VEL
LIN {X 0,Y 328.58,Z 775.917,A -85,B 0,C 180,E1 11803.904,E2 11803.904} C_VEL
LIN {X 0,Y 328.113,Z 780.822,A -85,B 0,C 180,E1 11800.175,E2 11800.175} C_VEL
LIN {X 0,Y 327.972,Z 784.055,A -85,B 0,C 180,E1 11796.476,E2 11796.476} C_VEL
LIN {X 0,Y 327.948,Z 785.807,A -85,B 0,C 180,E1 11793.146,E2 11793.146} C_VEL
LIN {X 0,Y 327.949,Z 786.333,A -85,B 0,C 180,E1 11789.476,E2 11789.476} C_VEL
LIN {X 0,Y 327.947,Z 785.518,A -85,B 0,C 180,E1 11786.154,E2 11786.154} C_VEL
LIN {X 0,Y 327.988,Z 783.449,A -85,B 0,C 180,E1 11782.644,E2 11782.644} C_VEL
LIN {X 0,Y 328.217,Z 779.515,A -85,B 0,C 180,E1 11778.758,E2 11778.758} C_VEL
LIN {X 0,Y 328.762,Z 774.563,A -85,B 0,C 180,E1 11775.199,E2 11775.199} C_VEL
LIN {X 0,Y 329.92,Z 767.373,A -85,B 0,C 180,E1 11771.262,E2 11771.262} C_VEL
LIN {X 0,Y 331.737,Z 758.888,A -85,B 0,C 180,E1 11767.495,E2 11767.495} C_VEL
LIN {X 0,Y 334.358,Z 748.423,A -85,B 0,C 180,E1 11763.732,E2 11763.732} C_VEL
LIN {X 0,Y 337.733,Z 736.647,A -85,B 0,C 180,E1 11760.16,E2 11760.16} C_VEL
LIN {X 0,Y 341.748,Z 723.576,A -85,B 0,C 180,E1 11756.832,E2 11756.832} C_VEL
LIN {X 0,Y 346.648,Z 708.32,A -85,B 0,C 180,E1 11753.547,E2 11753.547} C_VEL
LIN {X 0,Y 351.899,Z 692.282,A -85,B 0,C 180,E1 11750.609,E2 11750.609} C_VEL
LIN {X 0,Y 357.272,Z 675.421,A -85,B 0,C 180,E1 11748.022,E2 11748.022} C_VEL
LIN {X 0,Y 363,Z 656.931,A -85,B 0,C 180,E1 11745.605,E2 11745.605} C_VEL
LIN {X 0,Y 368.397,Z 638.333,A -85,B 0,C 180,E1 11743.561,E2 11743.561} C_VEL
LIN {X 0,Y 373.985,Z 617.442,A -85,B 0,C 180,E1 11741.649,E2 11741.649} C_VEL
LIN {X 0,Y 379.12,Z 596.319,A -85,B 0,C 180,E1 11740.053,E2 11740.053} C_VEL
LIN {X 0,Y 383.473,Z 575.311,A -85,B 0,C 180,E1 11738.778,E2 11738.778} C_VEL
LIN {X 0,Y 387.555,Z 552.182,A -85,B 0,C 180,E1 11737.66,E2 11737.66} C_VEL
LIN {X 0,Y 390.396,Z 532.048,A -85,B 0,C 180,E1 11736.914,E2 11736.914} C_VEL
LIN {X 0,Y 392.893,Z 507.439,A -85,B 0,C 180,E1 11736.249,E2 11736.249} C_VEL
LIN {X 0,Y 404.009,Z 313.051,A -85,B 0,C 180,E1 11732.325,E2 11732.325} C_VEL
LIN {X 0,Y 406.904,Z 262.581,A -85,B 0,C 180,E1 11731.312,E2 11731.312} C_VEL
LIN {X 0,Y 397.581,Z 248.016,A -85,B 0,C 180,E1 11728.748,E2 11728.748} C_VEL
LIN {X 0,Y 388.455,Z 234.768,A -85,B 0,C 180,E1 11725.949,E2 11725.949} C_VEL
LIN {X 0,Y 380.336,Z 223.908,A -85,B 0,C 180,E1 11723.142,E2 11723.142} C_VEL
LIN {X 0,Y 375.219,Z 217.421,A -85,B 0,C 180,E1 11721.166,E2 11721.166} C_VEL
LIN {X 0,Y 371.965,Z 213.347,A -85,B 0,C 180,E1 11719.797,E2 11719.797} C_VEL
LIN {X 0,Y 368.425,Z 209.008,A -85,B 0,C 180,E1 11718.185,E2 11718.185} C_VEL
LIN {X 0,Y 363.853,Z 203.589,A -85,B 0,C 180,E1 11715.868,E2 11715.868} C_VEL
LIN {X 0,Y 359.082,Z 198.041,A -85,B 0,C 180,E1 11713.035,E2 11713.035} C_VEL
LIN {X 0,Y 354.206,Z 192.791,A -85,B 0,C 180,E1 11709.423,E2 11709.423} C_VEL
LIN {X 0,Y 352.61,Z 191.36,A -85,B 0,C 180,E1 11707.986,E2 11707.986} C_VEL
LIN {X 0,Y 347.903,Z 186.729,A -85,B 0,C 180,E1 11701.152,E2 11701.152} C_VEL
LIN {X 0,Y 347.225,Z 186.157,A -85,B 0,C 180,E1 11697.854,E2 11697.854} C_VEL
LIN {X 0,Y 347.62,Z 187.552,A -85,B 0,C 180,E1 11694.056,E2 11694.056} C_VEL
LIN {X 0,Y 351.066,Z 191.534,A -85,B 0,C 180,E1 11688.167,E2 11688.167} C_VEL
LIN {X 0,Y 354.094,Z 195.843,A -85,B 0,C 180,E1 11685.11,E2 11685.11} C_VEL
LIN {X 0,Y 355.691,Z 197.453,A -85,B 0,C 180,E1 11683.841,E2 11683.841} C_VEL
LIN {X 0,Y 359.487,Z 202.348,A -85,B 0,C 180,E1 11681.177,E2 11681.177} C_VEL
LIN {X 0,Y 364.431,Z 208.862,A -85,B 0,C 180,E1 11678.303,E2 11678.303} C_VEL
LIN {X 0,Y 369.423,Z 215.491,A -85,B 0,C 180,E1 11675.835,E2 11675.835} C_VEL
LIN {X 0,Y 376.226,Z 224.837,A -85,B 0,C 180,E1 11672.927,E2 11672.927} C_VEL
LIN {X 0,Y 382.514,Z 233.934,A -85,B 0,C 180,E1 11670.566,E2 11670.566} C_VEL
LIN {X 0,Y 389.652,Z 244.478,A -85,B 0,C 180,E1 11668.175,E2 11668.175} C_VEL
LIN {X 0,Y 398.417,Z 258.621,A -85,B 0,C 180,E1 11665.534,E2 11665.534} C_VEL
LIN {X 0,Y 404.013,Z 268.396,A -85,B 0,C 180,E1 11663.981,E2 11663.981} C_VEL
LIN {X 0,Y 392.694,Z 495.893,A -85,B 0,C 180,E1 11659.701,E2 11659.701} C_VEL
LIN {X 0,Y 390.907,Z 522.44,A -85,B 0,C 180,E1 11659.138,E2 11659.138} C_VEL
LIN {X 0,Y 388.362,Z 544.255,A -85,B 0,C 180,E1 11658.477,E2 11658.477} C_VEL
LIN {X 0,Y 385.111,Z 564.682,A -85,B 0,C 180,E1 11657.614,E2 11657.614} C_VEL
LIN {X 0,Y 380.886,Z 586.3,A -85,B 0,C 180,E1 11656.427,E2 11656.427} C_VEL
LIN {X 0,Y 376.404,Z 605.701,A -85,B 0,C 180,E1 11655.099,E2 11655.099} C_VEL
LIN {X 0,Y 371.271,Z 624.765,A -85,B 0,C 180,E1 11653.477,E2 11653.477} C_VEL
LIN {X 0,Y 365.442,Z 644.269,A -85,B 0,C 180,E1 11651.46,E2 11651.46} C_VEL
LIN {X 0,Y 359.777,Z 661.817,A -85,B 0,C 180,E1 11649.264,E2 11649.264} C_VEL
LIN {X 0,Y 354.174,Z 677.87,A -85,B 0,C 180,E1 11646.829,E2 11646.829} C_VEL
LIN {X 0,Y 348.539,Z 693.467,A -85,B 0,C 180,E1 11643.998,E2 11643.998} C_VEL
LIN {X 0,Y 343.549,Z 707.223,A -85,B 0,C 180,E1 11641.006,E2 11641.006} C_VEL
LIN {X 0,Y 339.094,Z 719.52,A -85,B 0,C 180,E1 11637.766,E2 11637.766} C_VEL
LIN {X 0,Y 335.345,Z 730.41,A -85,B 0,C 180,E1 11634.296,E2 11634.296} C_VEL
LIN {X 0,Y 332.464,Z 739.652,A -85,B 0,C 180,E1 11630.722,E2 11630.722} C_VEL
LIN {X 0,Y 330.362,Z 747.343,A -85,B 0,C 180,E1 11626.982,E2 11626.982} C_VEL
LIN {X 0,Y 329.028,Z 753.438,A -85,B 0,C 180,E1 11623.174,E2 11623.174} C_VEL
LIN {X 0,Y 328.335,Z 757.985,A -85,B 0,C 180,E1 11619.369,E2 11619.369} C_VEL
LIN {X 0,Y 328.059,Z 760.741,A -85,B 0,C 180,E1 11615.772,E2 11615.772} C_VEL
LIN {X 0,Y 327.975,Z 762.289,A -85,B 0,C 180,E1 11612.096,E2 11612.096} C_VEL
LIN {X 0,Y 327.972,Z 762.313,A -85,B 0,C 180,E1 11611.892,E2 11611.892} C_VEL
LIN {X 0,Y 326.963,Z 762.525,A -85,B 0,C 180,E1 11610.547,E2 11610.547} C_VEL
LIN {X 0,Y 322.691,Z 762.539,A -85,B 0,C 180,E1 11608.193,E2 11608.193} C_VEL
LIN {X 0,Y 320.271,Z 762.174,A -85,B 0,C 180,E1 11606.443,E2 11606.443} C_VEL
LIN {X 0,Y 320.018,Z 761.921,A -85,B 0,C 180,E1 11605.744,E2 11605.744} C_VEL
LIN {X 0,Y 320.218,Z 759.486,A -85,B 0,C 180,E1 11601.742,E2 11601.742} C_VEL
LIN {X 0,Y 320.77,Z 755.764,A -85,B 0,C 180,E1 11597.946,E2 11597.946} C_VEL
LIN {X 0,Y 321.879,Z 750.406,A -85,B 0,C 180,E1 11594.136,E2 11594.136} C_VEL
LIN {X 0,Y 323.848,Z 743.134,A -85,B 0,C 180,E1 11590.147,E2 11590.147} C_VEL
LIN {X 0,Y 326.669,Z 734.4,A -85,B 0,C 180,E1 11586.362,E2 11586.362} C_VEL
LIN {X 0,Y 330.27,Z 724.164,A -85,B 0,C 180,E1 11582.798,E2 11582.798} C_VEL
LIN {X 0,Y 334.863,Z 711.98,A -85,B 0,C 180,E1 11579.298,E2 11579.298} C_VEL
LIN {X 0,Y 339.865,Z 699.071,A -85,B 0,C 180,E1 11576.22,E2 11576.22} C_VEL
LIN {X 0,Y 345.316,Z 684.675,A -85,B 0,C 180,E1 11573.384,E2 11573.384} C_VEL
LIN {X 0,Y 351.516,Z 667.907,A -85,B 0,C 180,E1 11570.633,E2 11570.633} C_VEL
LIN {X 0,Y 357.161,Z 651.859,A -85,B 0,C 180,E1 11568.436,E2 11568.436} C_VEL
LIN {X 0,Y 362.786,Z 634.334,A -85,B 0,C 180,E1 11566.449,E2 11566.449} C_VEL
LIN {X 0,Y 368.35,Z 615.451,A -85,B 0,C 180,E1 11564.671,E2 11564.671} C_VEL
LIN {X 0,Y 373.231,Z 596.695,A -85,B 0,C 180,E1 11563.227,E2 11563.227} C_VEL
LIN {X 0,Y 377.799,Z 576.213,A -85,B 0,C 180,E1 11561.956,E2 11561.956} C_VEL
LIN {X 0,Y 381.703,Z 555.322,A -85,B 0,C 180,E1 11560.934,E2 11560.934} C_VEL
LIN {X 0,Y 384.624,Z 534.906,A -85,B 0,C 180,E1 11560.188,E2 11560.188} C_VEL
LIN {X 0,Y 386.982,Z 511.318,A -85,B 0,C 180,E1 11559.576,E2 11559.576} C_VEL
LIN {X 0,Y 398.741,Z 285.948,A -85,B 0,C 180,E1 11555.295,E2 11555.295} C_VEL
LIN {X 0,Y 399.396,Z 272.026,A -85,B 0,C 180,E1 11555.004,E2 11555.004} C_VEL
LIN {X 0,Y 390.346,Z 256.659,A -85,B 0,C 180,E1 11552.311,E2 11552.311} C_VEL
LIN {X 0,Y 381.87,Z 243.467,A -85,B 0,C 180,E1 11549.488,E2 11549.488} C_VEL
LIN {X 0,Y 374.853,Z 233.166,A -85,B 0,C 180,E1 11546.837,E2 11546.837} C_VEL
LIN {X 0,Y 369.092,Z 224.949,A -85,B 0,C 180,E1 11544.358,E2 11544.358} C_VEL
LIN {X 0,Y 364.988,Z 219.476,A -85,B 0,C 180,E1 11542.382,E2 11542.382} C_VEL
LIN {X 0,Y 361.347,Z 214.528,A -85,B 0,C 180,E1 11540.405,E2 11540.405} C_VEL
LIN {X 0,Y 357.608,Z 209.6,A -85,B 0,C 180,E1 11538.081,E2 11538.081} C_VEL
LIN {X 0,Y 353.821,Z 204.473,A -85,B 0,C 180,E1 11535.237,E2 11535.237} C_VEL
LIN {X 0,Y 350.268,Z 200.061,A -85,B 0,C 180,E1 11531.777,E2 11531.777} C_VEL
LIN {X 0,Y 349.441,Z 198.791,A -85,B 0,C 180,E1 11530.719,E2 11530.719} C_VEL
LIN {X 0,Y 346.501,Z 194.915,A -85,B 0,C 180,E1 11523.971,E2 11523.971} C_VEL
LIN {X 0,Y 346.639,Z 194.484,A -85,B 0,C 180,E1 11520.661,E2 11520.661} C_VEL
LIN {X 0,Y 348.069,Z 196.171,A -85,B 0,C 180,E1 11516.707,E2 11516.707} C_VEL
LIN {X 0,Y 352.766,Z 200.321,A -85,B 0,C 180,E1 11511.114,E2 11511.114} C_VEL
LIN {X 0,Y 357.687,Z 205.789,A -85,B 0,C 180,E1 11507.304,E2 11507.304} C_VEL
LIN {X 0,Y 363.549,Z 212.771,A -85,B 0,C 180,E1 11503.791,E2 11503.791} C_VEL
LIN {X 0,Y 368.485,Z 218.792,A -85,B 0,C 180,E1 11501.326,E2 11501.326} C_VEL
LIN {X 0,Y 373.014,Z 224.546,A -85,B 0,C 180,E1 11499.32,E2 11499.32} C_VEL
LIN {X 0,Y 379.329,Z 232.643,A -85,B 0,C 180,E1 11496.834,E2 11496.834} C_VEL
LIN {X 0,Y 387.701,Z 244.424,A -85,B 0,C 180,E1 11493.915,E2 11493.915} C_VEL
LIN {X 0,Y 395.934,Z 256.652,A -85,B 0,C 180,E1 11491.368,E2 11491.368} C_VEL
LIN {X 0,Y 402.336,Z 266.955,A -85,B 0,C 180,E1 11489.547,E2 11489.547} C_VEL
LIN {X 0,Y 389.984,Z 475.308,A -85,B 0,C 180,E1 11485.354,E2 11485.354} C_VEL
LIN {X 0,Y 387.424,Z 514.63,A -85,B 0,C 180,E1 11484.518,E2 11484.518} C_VEL
LIN {X 0,Y 384.706,Z 537.324,A -85,B 0,C 180,E1 11483.845,E2 11483.845} C_VEL
LIN {X 0,Y 381.056,Z 560.503,A -85,B 0,C 180,E1 11482.906,E2 11482.906} C_VEL
LIN {X 0,Y 376.824,Z 582.449,A -85,B 0,C 180,E1 11481.756,E2 11481.756} C_VEL
LIN {X 0,Y 371.976,Z 603.475,A -85,B 0,C 180,E1 11480.361,E2 11480.361} C_VEL
LIN {X 0,Y 366.713,Z 623.952,A -85,B 0,C 180,E1 11478.714,E2 11478.714} C_VEL
LIN {X 0,Y 361.278,Z 642.811,A -85,B 0,C 180,E1 11476.876,E2 11476.876} C_VEL
LIN {X 0,Y 355.038,Z 662.983,A -85,B 0,C 180,E1 11474.525,E2 11474.525} C_VEL
LIN {X 0,Y 349.508,Z 679.865,A -85,B 0,C 180,E1 11472.189,E2 11472.189} C_VEL
LIN {X 0,Y 343.664,Z 697.039,A -85,B 0,C 180,E1 11469.363,E2 11469.363} C_VEL
LIN {X 0,Y 338.486,Z 712.284,A -85,B 0,C 180,E1 11466.421,E2 11466.421} C_VEL
LIN {X 0,Y 333.765,Z 726.134,A -85,B 0,C 180,E1 11463.243,E2 11463.243} C_VEL
LIN {X 0,Y 329.282,Z 740.053,A -85,B 0,C 180,E1 11459.465,E2 11459.465} C_VEL
LIN {X 0,Y 325.972,Z 751.307,A -85,B 0,C 180,E1 11455.82,E2 11455.82} C_VEL
LIN {X 0,Y 323.399,Z 761.151,A -85,B 0,C 180,E1 11451.95,E2 11451.95} C_VEL
LIN {X 0,Y 321.678,Z 769.264,A -85,B 0,C 180,E1 11448.108,E2 11448.108} C_VEL
LIN {X 0,Y 320.647,Z 775.596,A -85,B 0,C 180,E1 11444.261,E2 11444.261} C_VEL
LIN {X 0,Y 320.136,Z 780.514,A -85,B 0,C 180,E1 11440.436,E2 11440.436} C_VEL
LIN {X 0,Y 319.977,Z 783.759,A -85,B 0,C 180,E1 11436.639,E2 11436.639} C_VEL
LIN {X 0,Y 319.952,Z 785.515,A -85,B 0,C 180,E1 11433.225,E2 11433.225} C_VEL
LIN {X 0,Y 319.954,Z 786.042,A -85,B 0,C 180,E1 11429.463,E2 11429.463} C_VEL
LIN {X 0,Y 319.95,Z 785.225,A -85,B 0,C 180,E1 11426.058,E2 11426.058} C_VEL
LIN {X 0,Y 319.994,Z 783.151,A -85,B 0,C 180,E1 11422.459,E2 11422.459} C_VEL
LIN {X 0,Y 320.229,Z 779.406,A -85,B 0,C 180,E1 11418.639,E2 11418.639} C_VEL
LIN {X 0,Y 320.798,Z 774.518,A -85,B 0,C 180,E1 11415.008,E2 11415.008} C_VEL
LIN {X 0,Y 322.024,Z 767.417,A -85,B 0,C 180,E1 11410.973,E2 11410.973} C_VEL
LIN {X 0,Y 323.833,Z 759.404,A -85,B 0,C 180,E1 11407.298,E2 11407.298} C_VEL
LIN {X 0,Y 326.561,Z 749.148,A -85,B 0,C 180,E1 11403.448,E2 11403.448} C_VEL
LIN {X 0,Y 330.061,Z 737.642,A -85,B 0,C 180,E1 11399.811,E2 11399.811} C_VEL
LIN {X 0,Y 334.242,Z 724.654,A -85,B 0,C 180,E1 11396.4,E2 11396.4} C_VEL
LIN {X 0,Y 339.337,Z 709.669,A -85,B 0,C 180,E1 11393.053,E2 11393.053} C_VEL
LIN {X 0,Y 344.648,Z 694.131,A -85,B 0,C 180,E1 11390.124,E2 11390.124} C_VEL
LIN {X 0,Y 350.413,Z 677.028,A -85,B 0,C 180,E1 11387.406,E2 11387.406} C_VEL
LIN {X 0,Y 356.269,Z 659.16,A -85,B 0,C 180,E1 11384.992,E2 11384.992} C_VEL
LIN {X 0,Y 362.046,Z 640.061,A -85,B 0,C 180,E1 11382.844,E2 11382.844} C_VEL
LIN {X 0,Y 367.825,Z 619.581,A -85,B 0,C 180,E1 11380.916,E2 11380.916} C_VEL
LIN {X 0,Y 372.977,Z 599.264,A -85,B 0,C 180,E1 11379.342,E2 11379.342} C_VEL
LIN {X 0,Y 377.593,Z 578.378,A -85,B 0,C 180,E1 11378.024,E2 11378.024} C_VEL
LIN {X 0,Y 381.742,Z 556.571,A -85,B 0,C 180,E1 11376.919,E2 11376.919} C_VEL
LIN {X 0,Y 385.02,Z 534.627,A -85,B 0,C 180,E1 11376.074,E2 11376.074} C_VEL
LIN {X 0,Y 387.662,Z 511.263,A -85,B 0,C 180,E1 11375.408,E2 11375.408} C_VEL
LIN {X 0,Y 395.785,Z 375.024,A -85,B 0,C 180,E1 11372.626,E2 11372.626} C_VEL
LIN {X 0,Y 402.185,Z 266.66,A -85,B 0,C 180,E1 11370.433,E2 11370.433} C_VEL
LIN {X 0,Y 393.869,Z 253.602,A -85,B 0,C 180,E1 11368.051,E2 11368.051} C_VEL
LIN {X 0,Y 385.676,Z 241.501,A -85,B 0,C 180,E1 11365.449,E2 11365.449} C_VEL
LIN {X 0,Y 377.913,Z 230.911,A -85,B 0,C 180,E1 11362.682,E2 11362.682} C_VEL
LIN {X 0,Y 371.138,Z 222.031,A -85,B 0,C 180,E1 11359.925,E2 11359.925} C_VEL
LIN {X 0,Y 366.341,Z 216.207,A -85,B 0,C 180,E1 11357.717,E2 11357.717} C_VEL
LIN {X 0,Y 362.164,Z 211.137,A -85,B 0,C 180,E1 11355.533,E2 11355.533} C_VEL
LIN {X 0,Y 357.377,Z 205.544,A -85,B 0,C 180,E1 11352.605,E2 11352.605} C_VEL
LIN {X 0,Y 352.685,Z 200.188,A -85,B 0,C 180,E1 11348.97,E2 11348.97} C_VEL
LIN {X 0,Y 347.304,Z 195.226,A -85,B 0,C 180,E1 11342.145,E2 11342.145} C_VEL
LIN {X 0,Y 346.328,Z 194.085,A -85,B 0,C 180,E1 11338.676,E2 11338.676} C_VEL
LIN {X 0,Y 346.36,Z 194.821,A -85,B 0,C 180,E1 11335.364,E2 11335.364} C_VEL
LIN {X 0,Y 349.895,Z 199.38,A -85,B 0,C 180,E1 11328.377,E2 11328.377} C_VEL
LIN {X 0,Y 352.954,Z 203.742,A -85,B 0,C 180,E1 11325.229,E2 11325.229} C_VEL
LIN {X 0,Y 354.42,Z 205.345,A -85,B 0,C 180,E1 11324.034,E2 11324.034} C_VEL
LIN {X 0,Y 358.634,Z 210.997,A -85,B 0,C 180,E1 11321.046,E2 11321.046} C_VEL
LIN {X 0,Y 362.696,Z 216.36,A -85,B 0,C 180,E1 11318.661,E2 11318.661} C_VEL
LIN {X 0,Y 367.591,Z 222.989,A -85,B 0,C 180,E1 11316.176,E2 11316.176} C_VEL
LIN {X 0,Y 374.104,Z 232.135,A -85,B 0,C 180,E1 11313.32,E2 11313.32} C_VEL
LIN {X 0,Y 380.093,Z 240.981,A -85,B 0,C 180,E1 11311.008,E2 11311.008} C_VEL
LIN {X 0,Y 387.005,Z 251.435,A -85,B 0,C 180,E1 11308.628,E2 11308.628} C_VEL
LIN {X 0,Y 395.118,Z 264.733,A -85,B 0,C 180,E1 11306.11,E2 11306.11} C_VEL
LIN {X 0,Y 399.426,Z 272.349,A -85,B 0,C 180,E1 11304.866,E2 11304.866} C_VEL
LIN {X 0,Y 387.631,Z 499.588,A -85,B 0,C 180,E1 11300.565,E2 11300.565} C_VEL
LIN {X 0,Y 385.846,Z 523.513,A -85,B 0,C 180,E1 11300.041,E2 11300.041} C_VEL
LIN {X 0,Y 383.1,Z 545.677,A -85,B 0,C 180,E1 11299.352,E2 11299.352} C_VEL
LIN {X 0,Y 379.719,Z 566.089,A -85,B 0,C 180,E1 11298.476,E2 11298.476} C_VEL
LIN {X 0,Y 375.43,Z 587.015,A -85,B 0,C 180,E1 11297.31,E2 11297.31} C_VEL
LIN {X 0,Y 370.794,Z 606.318,A -85,B 0,C 180,E1 11295.976,E2 11295.976} C_VEL
LIN {X 0,Y 365.481,Z 625.303,A -85,B 0,C 180,E1 11294.344,E2 11294.344} C_VEL
LIN {X 0,Y 359.43,Z 644.737,A -85,B 0,C 180,E1 11292.312,E2 11292.312} C_VEL
LIN {X 0,Y 353.639,Z 661.952,A -85,B 0,C 180,E1 11290.137,E2 11290.137} C_VEL
LIN {X 0,Y 347.755,Z 678.115,A -85,B 0,C 180,E1 11287.659,E2 11287.659} C_VEL
LIN {X 0,Y 341.825,Z 693.776,A -85,B 0,C 180,E1 11284.776,E2 11284.776} C_VEL
LIN {X 0,Y 336.562,Z 707.573,A -85,B 0,C 180,E1 11281.723,E2 11281.723} C_VEL
LIN {X 0,Y 332.086,Z 719.252,A -85,B 0,C 180,E1 11278.601,E2 11278.601} C_VEL
LIN {X 0,Y 328.069,Z 730.245,A -85,B 0,C 180,E1 11275.063,E2 11275.063} C_VEL
LIN {X 0,Y 325.005,Z 739.443,A -85,B 0,C 180,E1 11271.474,E2 11271.474} C_VEL
LIN {X 0,Y 322.7,Z 747.154,A -85,B 0,C 180,E1 11267.676,E2 11267.676} C_VEL
LIN {X 0,Y 321.134,Z 753.742,A -85,B 0,C 180,E1 11263.504,E2 11263.504} C_VEL
LIN {X 0,Y 320.395,Z 758.193,A -85,B 0,C 180,E1 11259.701,E2 11259.701} C_VEL
LIN {X 0,Y 320.074,Z 761.035,A -85,B 0,C 180,E1 11255.917,E2 11255.917} C_VEL
LIN {X 0,Y 319.981,Z 762.58,A -85,B 0,C 180,E1 11252.149,E2 11252.149} C_VEL
LIN {X 0,Y 319.979,Z 762.675,A -85,B 0,C 180,E1 11248.568,E2 11248.568} C_VEL
LIN {X 0,Y 320.018,Z 761.921,A -85,B 0,C 180,E1 11245.744,E2 11245.744} C_VEL
LIN {X 0,Y 319.073,Z 761.387,A -85,B 0,C 180,E1 11244.367,E2 11244.367} C_VEL
LIN {X 0,Y 314.777,Z 760.031,A -85,B 0,C 180,E1 11241.86,E2 11241.86} C_VEL
LIN {X 0,Y 312.623,Z 758.6,A -85,B 0,C 180,E1 11240.077,E2 11240.077} C_VEL
LIN {X 0,Y 312.503,Z 757.992,A -85,B 0,C 180,E1 11239.472,E2 11239.472} C_VEL
LIN {X 0,Y 313.394,Z 753.448,A -85,B 0,C 180,E1 11235.591,E2 11235.591} C_VEL
LIN {X 0,Y 315.089,Z 746.968,A -85,B 0,C 180,E1 11231.499,E2 11231.499} C_VEL
LIN {X 0,Y 317.626,Z 739.116,A -85,B 0,C 180,E1 11227.611,E2 11227.611} C_VEL
LIN {X 0,Y 320.964,Z 729.829,A -85,B 0,C 180,E1 11223.945,E2 11223.945} C_VEL
LIN {X 0,Y 325.292,Z 718.672,A -85,B 0,C 180,E1 11220.34,E2 11220.34} C_VEL
LIN {X 0,Y 330.087,Z 706.888,A -85,B 0,C 180,E1 11217.167,E2 11217.167} C_VEL
LIN {X 0,Y 335.692,Z 692.906,A -85,B 0,C 180,E1 11214.074,E2 11214.074} C_VEL
LIN {X 0,Y 341.764,Z 677.512,A -85,B 0,C 180,E1 11211.24,E2 11211.24} C_VEL
LIN {X 0,Y 347.736,Z 661.8,A -85,B 0,C 180,E1 11208.82,E2 11208.82} C_VEL
LIN {X 0,Y 353.786,Z 644.522,A -85,B 0,C 180,E1 11206.628,E2 11206.628} C_VEL
LIN {X 0,Y 360.08,Z 625.002,A -85,B 0,C 180,E1 11204.584,E2 11204.584} C_VEL
LIN {X 0,Y 365.52,Z 606.236,A -85,B 0,C 180,E1 11202.97,E2 11202.97} C_VEL
LIN {X 0,Y 370.403,Z 586.529,A -85,B 0,C 180,E1 11201.608,E2 11201.608} C_VEL
LIN {X 0,Y 374.952,Z 564.808,A -85,B 0,C 180,E1 11200.409,E2 11200.409} C_VEL
LIN {X 0,Y 378.623,Z 543.192,A -85,B 0,C 180,E1 11199.501,E2 11199.501} C_VEL
LIN {X 0,Y 381.31,Z 521.198,A -85,B 0,C 180,E1 11198.848,E2 11198.848} C_VEL
LIN {X 0,Y 383.31,Z 491.829,A -85,B 0,C 180,E1 11198.233,E2 11198.233} C_VEL
LIN {X 0,Y 394.996,Z 276.188,A -85,B 0,C 180,E1 11194.123,E2 11194.123} C_VEL
LIN {X 0,Y 386.645,Z 262.002,A -85,B 0,C 180,E1 11191.535,E2 11191.535} C_VEL
LIN {X 0,Y 379.153,Z 250.105,A -85,B 0,C 180,E1 11188.941,E2 11188.941} C_VEL
LIN {X 0,Y 372.653,Z 240.326,A -85,B 0,C 180,E1 11186.406,E2 11186.406} C_VEL
LIN {X 0,Y 366.774,Z 231.814,A -85,B 0,C 180,E1 11183.795,E2 11183.795} C_VEL
LIN {X 0,Y 363.009,Z 226.683,A -85,B 0,C 180,E1 11181.914,E2 11181.914} C_VEL
LIN {X 0,Y 359.595,Z 221.94,A -85,B 0,C 180,E1 11179.999,E2 11179.999} C_VEL
LIN {X 0,Y 356.074,Z 217.178,A -85,B 0,C 180,E1 11177.739,E2 11177.739} C_VEL
LIN {X 0,Y 352.481,Z 212.203,A -85,B 0,C 180,E1 11174.96,E2 11174.96} C_VEL
LIN {X 0,Y 349.037,Z 207.761,A -85,B 0,C 180,E1 11171.484,E2 11171.484} C_VEL
LIN {X 0,Y 348.229,Z 206.568,A -85,B 0,C 180,E1 11170.422,E2 11170.422} C_VEL
LIN {X 0,Y 345.515,Z 202.818,A -85,B 0,C 180,E1 11163.817,E2 11163.817} C_VEL
LIN {X 0,Y 345.688,Z 202.475,A -85,B 0,C 180,E1 11160.497,E2 11160.497} C_VEL
LIN {X 0,Y 347.27,Z 204.367,A -85,B 0,C 180,E1 11156.369,E2 11156.369} C_VEL
LIN {X 0,Y 351.512,Z 208.136,A -85,B 0,C 180,E1 11151.33,E2 11151.33} C_VEL
LIN {X 0,Y 356.321,Z 213.556,A -85,B 0,C 180,E1 11147.522,E2 11147.522} C_VEL
LIN {X 0,Y 361.85,Z 220.308,A -85,B 0,C 180,E1 11144.124,E2 11144.124} C_VEL
LIN {X 0,Y 366.616,Z 226.242,A -85,B 0,C 180,E1 11141.681,E2 11141.681} C_VEL
LIN {X 0,Y 371.145,Z 232.12,A -85,B 0,C 180,E1 11139.623,E2 11139.623} C_VEL
LIN {X 0,Y 377.181,Z 240.06,A -85,B 0,C 180,E1 11137.189,E2 11137.189} C_VEL
LIN {X 0,Y 385.124,Z 251.422,A -85,B 0,C 180,E1 11134.348,E2 11134.348} C_VEL
LIN {X 0,Y 393.325,Z 263.872,A -85,B 0,C 180,E1 11131.741,E2 11131.741} C_VEL
LIN {X 0,Y 397.75,Z 271.295,A -85,B 0,C 180,E1 11130.429,E2 11130.429} C_VEL
LIN {X 0,Y 384.934,Z 480.054,A -85,B 0,C 180,E1 11126.211,E2 11126.211} C_VEL
LIN {X 0,Y 382.479,Z 515.439,A -85,B 0,C 180,E1 11125.447,E2 11125.447} C_VEL
LIN {X 0,Y 379.723,Z 537.697,A -85,B 0,C 180,E1 11124.783,E2 11124.783} C_VEL
LIN {X 0,Y 375.871,Z 561.223,A -85,B 0,C 180,E1 11123.822,E2 11123.822} C_VEL
LIN {X 0,Y 371.531,Z 582.941,A -85,B 0,C 180,E1 11122.676,E2 11122.676} C_VEL
LIN {X 0,Y 366.516,Z 603.849,A -85,B 0,C 180,E1 11121.278,E2 11121.278} C_VEL
LIN {X 0,Y 360.761,Z 625.232,A -85,B 0,C 180,E1 11119.532,E2 11119.532} C_VEL
LIN {X 0,Y 355.087,Z 644.15,A -85,B 0,C 180,E1 11117.657,E2 11117.657} C_VEL
LIN {X 0,Y 348.715,Z 663.777,A -85,B 0,C 180,E1 11115.321,E2 11115.321} C_VEL
LIN {X 0,Y 342.678,Z 681.429,A -85,B 0,C 180,E1 11112.83,E2 11112.83} C_VEL
LIN {X 0,Y 336.649,Z 698.22,A -85,B 0,C 180,E1 11109.98,E2 11109.98} C_VEL
LIN {X 0,Y 330.564,Z 715.098,A -85,B 0,C 180,E1 11106.573,E2 11106.573} C_VEL
LIN {X 0,Y 325.542,Z 729.388,A -85,B 0,C 180,E1 11103.14,E2 11103.14} C_VEL
LIN {X 0,Y 321.214,Z 742.091,A -85,B 0,C 180,E1 11099.459,E2 11099.459} C_VEL
LIN {X 0,Y 317.567,Z 753.932,A -85,B 0,C 180,E1 11095.352,E2 11095.352} C_VEL
LIN {X 0,Y 315.184,Z 762.906,A -85,B 0,C 180,E1 11091.591,E2 11091.591} C_VEL
LIN {X 0,Y 313.448,Z 770.867,A -85,B 0,C 180,E1 11087.448,E2 11087.448} C_VEL
LIN {X 0,Y 312.506,Z 776.896,A -85,B 0,C 180,E1 11083.506,E2 11083.506} C_VEL
LIN {X 0,Y 312.077,Z 781.24,A -85,B 0,C 180,E1 11079.59,E2 11079.59} C_VEL
LIN {X 0,Y 311.969,Z 783.826,A -85,B 0,C 180,E1 11076.256,E2 11076.256} C_VEL
LIN {X 0,Y 311.957,Z 785.509,A -85,B 0,C 180,E1 11072.388,E2 11072.388} C_VEL
LIN {X 0,Y 311.964,Z 785.68,A -85,B 0,C 180,E1 11068.898,E2 11068.898} C_VEL
LIN {X 0,Y 311.949,Z 784.786,A -85,B 0,C 180,E1 11065.588,E2 11065.588} C_VEL
LIN {X 0,Y 312.021,Z 782.421,A -85,B 0,C 180,E1 11061.709,E2 11061.709} C_VEL
LIN {X 0,Y 312.3,Z 778.684,A -85,B 0,C 180,E1 11057.989,E2 11057.989} C_VEL
LIN {X 0,Y 313.024,Z 773.37,A -85,B 0,C 180,E1 11054.039,E2 11054.039} C_VEL
LIN {X 0,Y 314.37,Z 766.351,A -85,B 0,C 180,E1 11050.105,E2 11050.105} C_VEL
LIN {X 0,Y 316.524,Z 757.758,A -85,B 0,C 180,E1 11046.151,E2 11046.151} C_VEL
LIN {X 0,Y 319.482,Z 747.534,A -85,B 0,C 180,E1 11042.335,E2 11042.335} C_VEL
LIN {X 0,Y 323.679,Z 734.647,A -85,B 0,C 180,E1 11038.324,E2 11038.324} C_VEL
LIN {X 0,Y 328.345,Z 721.379,A -85,B 0,C 180,E1 11034.864,E2 11034.864} C_VEL
LIN {X 0,Y 333.58,Z 706.655,A -85,B 0,C 180,E1 11031.652,E2 11031.652} C_VEL
LIN {X 0,Y 339.516,Z 690.243,A -85,B 0,C 180,E1 11028.615,E2 11028.615} C_VEL
LIN {X 0,Y 345.206,Z 673.965,A -85,B 0,C 180,E1 11026.079,E2 11026.079} C_VEL
LIN {X 0,Y 351.701,Z 654.579,A -85,B 0,C 180,E1 11023.538,E2 11023.538} C_VEL
LIN {X 0,Y 357.641,Z 635.793,A -85,B 0,C 180,E1 11021.477,E2 11021.477} C_VEL
LIN {X 0,Y 363.277,Z 616.006,A -85,B 0,C 180,E1 11019.683,E2 11019.683} C_VEL
LIN {X 0,Y 368.616,Z 595.412,A -85,B 0,C 180,E1 11018.132,E2 11018.132} C_VEL
LIN {X 0,Y 373.162,Z 574.891,A -85,B 0,C 180,E1 11016.883,E2 11016.883} C_VEL
LIN {X 0,Y 377.492,Z 551.79,A -85,B 0,C 180,E1 11015.768,E2 11015.768} C_VEL
LIN {X 0,Y 380.499,Z 531.763,A -85,B 0,C 180,E1 11015.03,E2 11015.03} C_VEL
LIN {X 0,Y 383.102,Z 507.425,A -85,B 0,C 180,E1 11014.371,E2 11014.371} C_VEL
LIN {X 0,Y 395.042,Z 313.347,A -85,B 0,C 180,E1 11010.419,E2 11010.419} C_VEL
LIN {X 0,Y 397.678,Z 270.931,A -85,B 0,C 180,E1 11009.565,E2 11009.565} C_VEL
LIN {X 0,Y 388.644,Z 256.686,A -85,B 0,C 180,E1 11006.84,E2 11006.84} C_VEL
LIN {X 0,Y 379.907,Z 243.864,A -85,B 0,C 180,E1 11003.869,E2 11003.869} C_VEL
LIN {X 0,Y 372.499,Z 233.844,A -85,B 0,C 180,E1 11000.998,E2 11000.998} C_VEL
LIN {X 0,Y 367.506,Z 227.45,A -85,B 0,C 180,E1 10998.808,E2 10998.808} C_VEL
LIN {X 0,Y 364.284,Z 223.395,A -85,B 0,C 180,E1 10997.243,E2 10997.243} C_VEL
LIN {X 0,Y 360.351,Z 218.552,A -85,B 0,C 180,E1 10995.118,E2 10995.118} C_VEL
LIN {X 0,Y 355.925,Z 213.238,A -85,B 0,C 180,E1 10992.327,E2 10992.327} C_VEL
LIN {X 0,Y 350.996,Z 207.577,A -85,B 0,C 180,E1 10988.353,E2 10988.353} C_VEL
LIN {X 0,Y 345.938,Z 202.66,A -85,B 0,C 180,E1 10981.159,E2 10981.159} C_VEL
LIN {X 0,Y 345.286,Z 202.035,A -85,B 0,C 180,E1 10978.008,E2 10978.008} C_VEL
LIN {X 0,Y 345.582,Z 203.329,A -85,B 0,C 180,E1 10974.354,E2 10974.354} C_VEL
LIN {X 0,Y 348.726,Z 207.224,A -85,B 0,C 180,E1 10968.589,E2 10968.589} C_VEL
LIN {X 0,Y 352.005,Z 211.816,A -85,B 0,C 180,E1 10965.188,E2 10965.188} C_VEL
LIN {X 0,Y 353.153,Z 213.239,A -85,B 0,C 180,E1 10964.228,E2 10964.228} C_VEL
LIN {X 0,Y 357.184,Z 218.764,A -85,B 0,C 180,E1 10961.306,E2 10961.306} C_VEL
LIN {X 0,Y 361.04,Z 223.959,A -85,B 0,C 180,E1 10958.983,E2 10958.983} C_VEL
LIN {X 0,Y 365.773,Z 230.486,A -85,B 0,C 180,E1 10956.521,E2 10956.521} C_VEL
LIN {X 0,Y 372.087,Z 239.561,A -85,B 0,C 180,E1 10953.68,E2 10953.68} C_VEL
LIN {X 0,Y 377.792,Z 248.173,A -85,B 0,C 180,E1 10951.421,E2 10951.421} C_VEL
LIN {X 0,Y 384.485,Z 258.562,A -85,B 0,C 180,E1 10949.052,E2 10949.052} C_VEL
LIN {X 0,Y 391.988,Z 271.074,A -85,B 0,C 180,E1 10946.654,E2 10946.654} C_VEL
LIN {X 0,Y 394.932,Z 276.386,A -85,B 0,C 180,E1 10945.77,E2 10945.77} C_VEL
LIN {X 0,Y 382.699,Z 502.432,A -85,B 0,C 180,E1 10941.468,E2 10941.468} C_VEL
LIN {X 0,Y 380.828,Z 525.106,A -85,B 0,C 180,E1 10940.954,E2 10940.954} C_VEL
LIN {X 0,Y 377.767,Z 548.112,A -85,B 0,C 180,E1 10940.212,E2 10940.212} C_VEL
LIN {X 0,Y 374.091,Z 569.285,A -85,B 0,C 180,E1 10939.274,E2 10939.274} C_VEL
LIN {X 0,Y 369.718,Z 589.221,A -85,B 0,C 180,E1 10938.123,E2 10938.123} C_VEL
LIN {X 0,Y 364.424,Z 609.852,A -85,B 0,C 180,E1 10936.64,E2 10936.64} C_VEL
LIN {X 0,Y 358.879,Z 628.854,A -85,B 0,C 180,E1 10934.955,E2 10934.955} C_VEL
LIN {X 0,Y 352.831,Z 647.163,A -85,B 0,C 180,E1 10932.962,E2 10932.962} C_VEL
LIN {X 0,Y 346.24,Z 665.62,A -85,B 0,C 180,E1 10930.521,E2 10930.521} C_VEL
LIN {X 0,Y 340.429,Z 680.982,A -85,B 0,C 180,E1 10928.08,E2 10928.08} C_VEL
LIN {X 0,Y 334.498,Z 695.786,A -85,B 0,C 180,E1 10925.232,E2 10925.232} C_VEL
LIN {X 0,Y 328.781,Z 709.954,A -85,B 0,C 180,E1 10921.947,E2 10921.947} C_VEL
LIN {X 0,Y 323.997,Z 722.009,A -85,B 0,C 180,E1 10918.576,E2 10918.576} C_VEL
LIN {X 0,Y 319.94,Z 732.55,A -85,B 0,C 180,E1 10914.953,E2 10914.953} C_VEL
LIN {X 0,Y 316.726,Z 741.7,A -85,B 0,C 180,E1 10911.092,E2 10911.092} C_VEL
LIN {X 0,Y 314.496,Z 749.12,A -85,B 0,C 180,E1 10907.197,E2 10907.197} C_VEL
LIN {X 0,Y 313.093,Z 754.768,A -85,B 0,C 180,E1 10903.293,E2 10903.293} C_VEL
LIN {X 0,Y 312.319,Z 759.249,A -85,B 0,C 180,E1 10899.025,E2 10899.025} C_VEL
LIN {X 0,Y 312.056,Z 761.757,A -85,B 0,C 180,E1 10895.331,E2 10895.331} C_VEL
LIN {X 0,Y 311.98,Z 762.955,A -85,B 0,C 180,E1 10891.469,E2 10891.469} C_VEL
LIN {X 0,Y 311.985,Z 762.903,A -85,B 0,C 180,E1 10887.98,E2 10887.98} C_VEL
LIN {X 0,Y 312.077,Z 761.493,A -85,B 0,C 180,E1 10884.116,E2 10884.116} C_VEL
LIN {X 0,Y 312.384,Z 758.817,A -85,B 0,C 180,E1 10880.343,E2 10880.343} C_VEL
LIN {X 0,Y 312.503,Z 757.992,A -85,B 0,C 180,E1 10879.472,E2 10879.472} C_VEL
LIN {X 0,Y 311.751,Z 756.615,A -85,B 0,C 180,E1 10878.079,E2 10878.079} C_VEL
LIN {X 0,Y 306.503,Z 752.354,A -85,B 0,C 180,E1 10874.227,E2 10874.227} C_VEL
LIN {X 0,Y 306.324,Z 750.737,A -85,B 0,C 180,E1 10873.119,E2 10873.119} C_VEL
LIN {X 0,Y 308.78,Z 742.985,A -85,B 0,C 180,E1 10868.737,E2 10868.737} C_VEL
LIN {X 0,Y 312.088,Z 734.108,A -85,B 0,C 180,E1 10864.78,E2 10864.78} C_VEL
LIN {X 0,Y 316.246,Z 723.714,A -85,B 0,C 180,E1 10861.071,E2 10861.071} C_VEL
LIN {X 0,Y 321.457,Z 711.319,A -85,B 0,C 180,E1 10857.45,E2 10857.45} C_VEL
LIN {X 0,Y 327.063,Z 698.195,A -85,B 0,C 180,E1 10854.276,E2 10854.276} C_VEL
LIN {X 0,Y 333.136,Z 683.618,A -85,B 0,C 180,E1 10851.372,E2 10851.372} C_VEL
LIN {X 0,Y 339.538,Z 667.634,A -85,B 0,C 180,E1 10848.73,E2 10848.73} C_VEL
LIN {X 0,Y 345.874,Z 650.921,A -85,B 0,C 180,E1 10846.424,E2 10846.424} C_VEL
LIN {X 0,Y 352.007,Z 633.13,A -85,B 0,C 180,E1 10844.41,E2 10844.41} C_VEL
LIN {X 0,Y 358.018,Z 613.912,A -85,B 0,C 180,E1 10842.619,E2 10842.619} C_VEL
LIN {X 0,Y 363.278,Z 594.948,A -85,B 0,C 180,E1 10841.172,E2 10841.172} C_VEL
LIN {X 0,Y 367.895,Z 575.217,A -85,B 0,C 180,E1 10839.969,E2 10839.969} C_VEL
LIN {X 0,Y 371.978,Z 554.418,A -85,B 0,C 180,E1 10838.963,E2 10838.963} C_VEL
LIN {X 0,Y 375.049,Z 534.2,A -85,B 0,C 180,E1 10838.232,E2 10838.232} C_VEL
LIN {X 0,Y 377.499,Z 510.893,A -85,B 0,C 180,E1 10837.631,E2 10837.631} C_VEL
LIN {X 0,Y 390.345,Z 285.02,A -85,B 0,C 180,E1 10833.295,E2 10833.295} C_VEL
LIN {X 0,Y 390.522,Z 280.205,A -85,B 0,C 180,E1 10833.176,E2 10833.176} C_VEL
LIN {X 0,Y 382.989,Z 267.286,A -85,B 0,C 180,E1 10830.733,E2 10830.733} C_VEL
LIN {X 0,Y 376.379,Z 256.597,A -85,B 0,C 180,E1 10828.35,E2 10828.35} C_VEL
LIN {X 0,Y 370.304,Z 247.236,A -85,B 0,C 180,E1 10825.896,E2 10825.896} C_VEL
LIN {X 0,Y 364.541,Z 238.731,A -85,B 0,C 180,E1 10823.248,E2 10823.248} C_VEL
LIN {X 0,Y 361.054,Z 233.884,A -85,B 0,C 180,E1 10821.441,E2 10821.441} C_VEL
LIN {X 0,Y 357.862,Z 229.349,A -85,B 0,C 180,E1 10819.59,E2 10819.59} C_VEL
LIN {X 0,Y 354.434,Z 224.628,A -85,B 0,C 180,E1 10817.315,E2 10817.315} C_VEL
LIN {X 0,Y 351.15,Z 219.931,A -85,B 0,C 180,E1 10814.68,E2 10814.68} C_VEL
LIN {X 0,Y 347.752,Z 215.328,A -85,B 0,C 180,E1 10811.107,E2 10811.107} C_VEL
LIN {X 0,Y 346.904,Z 214.258,A -85,B 0,C 180,E1 10809.959,E2 10809.959} C_VEL
LIN {X 0,Y 344.527,Z 210.721,A -85,B 0,C 180,E1 10803.661,E2 10803.661} C_VEL
LIN {X 0,Y 344.711,Z 210.421,A -85,B 0,C 180,E1 10800.499,E2 10800.499} C_VEL
LIN {X 0,Y 346.287,Z 212.346,A -85,B 0,C 180,E1 10796.358,E2 10796.358} C_VEL
LIN {X 0,Y 350.263,Z 215.949,A -85,B 0,C 180,E1 10791.546,E2 10791.546} C_VEL
LIN {X 0,Y 355.539,Z 222.163,A -85,B 0,C 180,E1 10787.329,E2 10787.329} C_VEL
LIN {X 0,Y 360.297,Z 228.035,A -85,B 0,C 180,E1 10784.385,E2 10784.385} C_VEL
LIN {X 0,Y 364.91,Z 233.9,A -85,B 0,C 180,E1 10781.964,E2 10781.964} C_VEL
LIN {X 0,Y 370.304,Z 240.977,A -85,B 0,C 180,E1 10779.492,E2 10779.492} C_VEL
LIN {X 0,Y 376.699,Z 249.843,A -85,B 0,C 180,E1 10776.911,E2 10776.911} C_VEL
LIN {X 0,Y 384.276,Z 260.963,A -85,B 0,C 180,E1 10774.204,E2 10774.204} C_VEL
LIN {X 0,Y 393.114,Z 274.947,A -85,B 0,C 180,E1 10771.393,E2 10771.393} C_VEL
LIN {X 0,Y 393.236,Z 276.062,A -85,B 0,C 180,E1 10771.324,E2 10771.324} C_VEL
LIN {X 0,Y 379.962,Z 485.002,A -85,B 0,C 180,E1 10767.087,E2 10767.087} C_VEL
LIN {X 0,Y 377.554,Z 516.974,A -85,B 0,C 180,E1 10766.38,E2 10766.38} C_VEL
LIN {X 0,Y 374.703,Z 539.073,A -85,B 0,C 180,E1 10765.712,E2 10765.712} C_VEL
LIN {X 0,Y 370.843,Z 561.656,A -85,B 0,C 180,E1 10764.778,E2 10764.778} C_VEL
LIN {X 0,Y 366.337,Z 583.417,A -85,B 0,C 180,E1 10763.623,E2 10763.623} C_VEL
LIN {X 0,Y 360.888,Z 605.249,A -85,B 0,C 180,E1 10762.147,E2 10762.147} C_VEL
LIN {X 0,Y 354.687,Z 627.174,A -85,B 0,C 180,E1 10760.315,E2 10760.315} C_VEL
LIN {X 0,Y 348.71,Z 646.321,A -85,B 0,C 180,E1 10758.377,E2 10758.377} C_VEL
LIN {X 0,Y 342.462,Z 664.575,A -85,B 0,C 180,E1 10756.147,E2 10756.147} C_VEL
LIN {X 0,Y 336.038,Z 682.451,A -85,B 0,C 180,E1 10753.566,E2 10753.566} C_VEL
LIN {X 0,Y 329.901,Z 698.786,A -85,B 0,C 180,E1 10750.739,E2 10750.739} C_VEL
LIN {X 0,Y 323.855,Z 714.728,A -85,B 0,C 180,E1 10747.459,E2 10747.459} C_VEL
LIN {X 0,Y 318.533,Z 729.031,A -85,B 0,C 180,E1 10743.967,E2 10743.967} C_VEL
LIN {X 0,Y 313.932,Z 741.746,A -85,B 0,C 180,E1 10740.212,E2 10740.212} C_VEL
LIN {X 0,Y 310.037,Z 753.6,A -85,B 0,C 180,E1 10736.014,E2 10736.014} C_VEL
LIN {X 0,Y 307.474,Z 762.58,A -85,B 0,C 180,E1 10732.161,E2 10732.161} C_VEL
LIN {X 0,Y 305.591,Z 770.553,A -85,B 0,C 180,E1 10727.912,E2 10727.912} C_VEL
LIN {X 0,Y 304.564,Z 776.588,A -85,B 0,C 180,E1 10723.866,E2 10723.866} C_VEL
LIN {X 0,Y 304.09,Z 780.941,A -85,B 0,C 180,E1 10719.844,E2 10719.844} C_VEL
LIN {X 0,Y 303.977,Z 783.531,A -85,B 0,C 180,E1 10716.421,E2 10716.421} C_VEL
LIN {X 0,Y 303.962,Z 785.218,A -85,B 0,C 180,E1 10712.451,E2 10712.451} C_VEL
LIN {X 0,Y 303.969,Z 785.389,A -85,B 0,C 180,E1 10708.869,E2 10708.869} C_VEL
LIN {X 0,Y 303.952,Z 784.494,A -85,B 0,C 180,E1 10705.472,E2 10705.472} C_VEL
LIN {X 0,Y 304.025,Z 782.121,A -85,B 0,C 180,E1 10701.49,E2 10701.49} C_VEL
LIN {X 0,Y 304.338,Z 778.38,A -85,B 0,C 180,E1 10697.67,E2 10697.67} C_VEL
LIN {X 0,Y 305.122,Z 773.085,A -85,B 0,C 180,E1 10693.632,E2 10693.632} C_VEL
LIN {X 0,Y 306.594,Z 766.029,A -85,B 0,C 180,E1 10689.578,E2 10689.578} C_VEL
LIN {X 0,Y 308.917,Z 757.423,A -85,B 0,C 180,E1 10685.526,E2 10685.526} C_VEL
LIN {X 0,Y 312.019,Z 747.387,A -85,B 0,C 180,E1 10681.689,E2 10681.689} C_VEL
LIN {X 0,Y 316.323,Z 734.95,A -85,B 0,C 180,E1 10677.712,E2 10677.712} C_VEL
LIN {X 0,Y 320.934,Z 722.467,A -85,B 0,C 180,E1 10674.368,E2 10674.368} C_VEL
LIN {X 0,Y 326.7,Z 707.141,A -85,B 0,C 180,E1 10670.917,E2 10670.917} C_VEL
LIN {X 0,Y 332.712,Z 691.389,A -85,B 0,C 180,E1 10667.922,E2 10667.922} C_VEL
LIN {X 0,Y 339.019,Z 674.101,A -85,B 0,C 180,E1 10665.182,E2 10665.182} C_VEL
LIN {X 0,Y 345.792,Z 654.779,A -85,B 0,C 180,E1 10662.619,E2 10662.619} C_VEL
LIN {X 0,Y 352.21,Z 635.282,A -85,B 0,C 180,E1 10660.467,E2 10660.467} C_VEL
LIN {X 0,Y 358.001,Z 615.638,A -85,B 0,C 180,E1 10658.685,E2 10658.685} C_VEL
LIN {X 0,Y 363.59,Z 594.69,A -85,B 0,C 180,E1 10657.111,E2 10657.111} C_VEL
